LIN {X 0,Y 233.314,Z 747.017,A -85,B 0,C 180,E1 -22157.757,E2 -22157.757} C_VEL
LIN {X 0,Y 234.312,Z 748.351,A -85,B 0,C 180,E1 -22158.64,E2 -22158.64} C_VEL
LIN {X 0,Y 237.807,Z 753.166,A -85,B 0,C 180,E1 -22161.415,E2 -22161.415} C_VEL
LIN {X 0,Y 240.661,Z 757.385,A -85,B 0,C 180,E1 -22163.417,E2 -22163.417} C_VEL
LIN {X 0,Y 245.508,Z 764.562,A -85,B 0,C 180,E1 -22166.397,E2 -22166.397} C_VEL
LIN {X 0,Y 250.605,Z 772.878,A -85,B 0,C 180,E1 -22169.16,E2 -22169.16} C_VEL
LIN {X 0,Y 260.08,Z 786.969,A -85,B 0,C 180,E1 -22173.436,E2 -22173.436} C_VEL
LIN {X 0,Y 267.5,Z 795.645,A -85,B 0,C 180,E1 -22176.179,E2 -22176.179} C_VEL
LIN {X 0,Y 274.994,Z 803.198,A -85,B 0,C 180,E1 -22178.59,E2 -22178.59} C_VEL
LIN {X 0,Y 289.384,Z 815.503,A -85,B 0,C 180,E1 -22182.579,E2 -22182.579} C_VEL
LIN {X 0,Y 297.408,Z 822.094,A -85,B 0,C 180,E1 -22184.884,E2 -22184.884} C_VEL
LIN {X 0,Y 304.266,Z 827.849,A -85,B 0,C 180,E1 -22187.056,E2 -22187.056} C_VEL
LIN {X 0,Y 310.212,Z 832.821,A -85,B 0,C 180,E1 -22189.111,E2 -22189.111} C_VEL
LIN {X 0,Y 316.754,Z 838.584,A -85,B 0,C 180,E1 -22191.56,E2 -22191.56} C_VEL
LIN {X 0,Y 321.993,Z 842.915,A -85,B 0,C 180,E1 -22193.61,E2 -22193.61} C_VEL
LIN {X 0,Y 327.654,Z 847.59,A -85,B 0,C 180,E1 -22195.919,E2 -22195.919} C_VEL
LIN {X 0,Y 333.978,Z 853.067,A -85,B 0,C 180,E1 -22198.672,E2 -22198.672} C_VEL
LIN {X 0,Y 338.981,Z 856.943,A -85,B 0,C 180,E1 -22200.959,E2 -22200.959} C_VEL
LIN {X 0,Y 343.44,Z 860.757,A -85,B 0,C 180,E1 -22203.147,E2 -22203.147} C_VEL
LIN {X 0,Y 347.97,Z 863.872,A -85,B 0,C 180,E1 -22205.496,E2 -22205.496} C_VEL
LIN {X 0,Y 352.286,Z 867.651,A -85,B 0,C 180,E1 -22208.002,E2 -22208.002} C_VEL
LIN {X 0,Y 356.283,Z 870.579,A -85,B 0,C 180,E1 -22210.538,E2 -22210.538} C_VEL
LIN {X 0,Y 359.499,Z 872.581,A -85,B 0,C 180,E1 -22212.766,E2 -22212.766} C_VEL
LIN {X 0,Y 362.492,Z 875.444,A -85,B 0,C 180,E1 -22215.247,E2 -22215.247} C_VEL
LIN {X 0,Y 365.132,Z 877.452,A -85,B 0,C 180,E1 -22217.777,E2 -22217.777} C_VEL
LIN {X 0,Y 367.207,Z 878.655,A -85,B 0,C 180,E1 -22220.082,E2 -22220.082} C_VEL
LIN {X 0,Y 368.794,Z 879.391,A -85,B 0,C 180,E1 -22222.334,E2 -22222.334} C_VEL
LIN {X 0,Y 369.977,Z 879.911,A -85,B 0,C 180,E1 -22224.55,E2 -22224.55} C_VEL
LIN {X 0,Y 370.787,Z 880.342,A -85,B 0,C 180,E1 -22226.74,E2 -22226.74} C_VEL
LIN {X 0,Y 371.141,Z 880.49,A -85,B 0,C 180,E1 -22228.915,E2 -22228.915} C_VEL
LIN {X 0,Y 371.14,Z 880.491,A -85,B 0,C 180,E1 -22231.085,E2 -22231.085} C_VEL
LIN {X 0,Y 370.787,Z 880.343,A -85,B 0,C 180,E1 -22233.26,E2 -22233.26} C_VEL
LIN {X 0,Y 369.977,Z 879.915,A -85,B 0,C 180,E1 -22235.45,E2 -22235.45} C_VEL
LIN {X 0,Y 368.777,Z 879.363,A -85,B 0,C 180,E1 -22237.7,E2 -22237.7} C_VEL
LIN {X 0,Y 366.736,Z 878.408,A -85,B 0,C 180,E1 -22240.449,E2 -22240.449} C_VEL
LIN {X 0,Y 364.408,Z 876.944,A -85,B 0,C 180,E1 -22242.986,E2 -22242.986} C_VEL
LIN {X 0,Y 361.479,Z 874.571,A -85,B 0,C 180,E1 -22245.627,E2 -22245.627} C_VEL
LIN {X 0,Y 358.848,Z 871.974,A -85,B 0,C 180,E1 -22247.72,E2 -22247.72} C_VEL
LIN {X 0,Y 355.4,Z 869.953,A -85,B 0,C 180,E1 -22250.056,E2 -22250.056} C_VEL
LIN {X 0,Y 351.316,Z 866.844,A -85,B 0,C 180,E1 -22252.572,E2 -22252.572} C_VEL
LIN {X 0,Y 347.804,Z 863.747,A -85,B 0,C 180,E1 -22254.592,E2 -22254.592} C_VEL
LIN {X 0,Y 342.734,Z 860.245,A -85,B 0,C 180,E1 -22257.204,E2 -22257.204} C_VEL
LIN {X 0,Y 337.022,Z 855.328,A -85,B 0,C 180,E1 -22259.96,E2 -22259.96} C_VEL
LIN {X 0,Y 331.892,Z 851.318,A -85,B 0,C 180,E1 -22262.255,E2 -22262.255} C_VEL
LIN {X 0,Y 326.884,Z 847.01,A -85,B 0,C 180,E1 -22264.4,E2 -22264.4} C_VEL
LIN {X 0,Y 321.053,Z 842.045,A -85,B 0,C 180,E1 -22266.767,E2 -22266.767} C_VEL
LIN {X 0,Y 313.987,Z 836.199,A -85,B 0,C 180,E1 -22269.498,E2 -22269.498} C_VEL
LIN {X 0,Y 307.168,Z 830.349,A -85,B 0,C 180,E1 -22271.968,E2 -22271.968} C_VEL
LIN {X 0,Y 300.834,Z 824.92,A -85,B 0,C 180,E1 -22274.041,E2 -22274.041} C_VEL
LIN {X 0,Y 294.494,Z 819.582,A -85,B 0,C 180,E1 -22275.97,E2 -22275.97} C_VEL
LIN {X 0,Y 286.718,Z 813.265,A -85,B 0,C 180,E1 -22278.147,E2 -22278.147} C_VEL
LIN {X 0,Y 276.516,Z 804.475,A -85,B 0,C 180,E1 -22280.962,E2 -22280.962} C_VEL
LIN {X 0,Y 269.019,Z 797.351,A -85,B 0,C 180,E1 -22283.303,E2 -22283.303} C_VEL
LIN {X 0,Y 259.248,Z 785.918,A -85,B 0,C 180,E1 -22286.898,E2 -22286.898} C_VEL
LIN {X 0,Y 247.028,Z 766.992,A -85,B 0,C 180,E1 -22292.742,E2 -22292.742} C_VEL
LIN {X 0,Y 241.698,Z 758.869,A -85,B 0,C 180,E1 -22295.909,E2 -22295.909} C_VEL
LIN {X 0,Y 238.957,Z 754.892,A -85,B 0,C 180,E1 -22297.749,E2 -22297.749} C_VEL
LIN {X 0,Y 236.64,Z 751.543,A -85,B 0,C 180,E1 -22299.463,E2 -22299.463} C_VEL
LIN {X 0,Y 233.435,Z 747.121,A -85,B 0,C 180,E1 -22302.139,E2 -22302.139} C_VEL
LIN {X 0,Y 230.685,Z 743.267,A -85,B 0,C 180,E1 -22304.879,E2 -22304.879} C_VEL
LIN {X 0,Y 230.017,Z 742.388,A -85,B 0,C 180,E1 -22305.626,E2 -22305.626} C_VEL
LIN {X 0,Y 227.655,Z 739.605,A -85,B 0,C 180,E1 -22308.65,E2 -22308.65} C_VEL
LIN {X 0,Y 226.765,Z 737.637,A -85,B 0,C 180,E1 -22310.215,E2 -22310.215} C_VEL
LIN {X 0,Y 224.026,Z 734.193,A -85,B 0,C 180,E1 -22320,E2 -22320} C_VEL
LIN {X 0,Y 226.883,Z 737.813,A -85,B 0,C 180,E1 -22329.585,E2 -22329.585} C_VEL
LIN {X 0,Y 228.698,Z 741.176,A -85,B 0,C 180,E1 -22332.423,E2 -22332.423} C_VEL
LIN {X 0,Y 230.599,Z 743.15,A -85,B 0,C 180,E1 -22334.619,E2 -22334.619} C_VEL
LIN {X 0,Y 233.265,Z 746.992,A -85,B 0,C 180,E1 -22337.309,E2 -22337.309} C_VEL
LIN {X 0,Y 234.487,Z 748.68,A -85,B 0,C 180,E1 -22338.391,E2 -22338.391} C_VEL
LIN {X 0,Y 237.725,Z 753.072,A -85,B 0,C 180,E1 -22340.949,E2 -22340.949} C_VEL
LIN {X 0,Y 240.892,Z 757.691,A -85,B 0,C 180,E1 -22343.16,E2 -22343.16} C_VEL
LIN {X 0,Y 245.663,Z 764.824,A -85,B 0,C 180,E1 -22346.08,E2 -22346.08} C_VEL
LIN {X 0,Y 250.2,Z 773.785,A -85,B 0,C 180,E1 -22348.638,E2 -22348.638} C_VEL
LIN {X 0,Y 254.973,Z 784.136,A -85,B 0,C 180,E1 -22351.084,E2 -22351.084} C_VEL
LIN {X 0,Y 259.68,Z 795.604,A -85,B 0,C 180,E1 -22353.32,E2 -22353.32} C_VEL
LIN {X 0,Y 252.558,Z 888.891,A -85,B 0,C 180,E1 -22355.604,E2 -22355.604} C_VEL
LIN {X 0,Y 250.81,Z 902.408,A -85,B 0,C 180,E1 -22356.075,E2 -22356.075} C_VEL
LIN {X 0,Y 248.59,Z 914.617,A -85,B 0,C 180,E1 -22356.608,E2 -22356.608} C_VEL
LIN {X 0,Y 245.71,Z 927.15,A -85,B 0,C 180,E1 -22357.298,E2 -22357.298} C_VEL
LIN {X 0,Y 243.03,Z 937.334,A -85,B 0,C 180,E1 -22358.001,E2 -22358.001} C_VEL
LIN {X 0,Y 238.986,Z 950.564,A -85,B 0,C 180,E1 -22359.14,E2 -22359.14} C_VEL
LIN {X 0,Y 235.019,Z 961.857,A -85,B 0,C 180,E1 -22360.312,E2 -22360.312} C_VEL
LIN {X 0,Y 230.1,Z 974.284,A -85,B 0,C 180,E1 -22361.886,E2 -22361.886} C_VEL
LIN {X 0,Y 226.127,Z 983.479,A -85,B 0,C 180,E1 -22363.256,E2 -22363.256} C_VEL
LIN {X 0,Y 220.297,Z 995.568,A -85,B 0,C 180,E1 -22365.426,E2 -22365.426} C_VEL
LIN {X 0,Y 215.559,Z 1004.833,A -85,B 0,C 180,E1 -22367.429,E2 -22367.429} C_VEL
LIN {X 0,Y 213.299,Z 1009.008,A -85,B 0,C 180,E1 -22368.464,E2 -22368.464} C_VEL
LIN {X 0,Y 210.589,Z 1013.057,A -85,B 0,C 180,E1 -22369.393,E2 -22369.393} C_VEL
LIN {X 0,Y 199.902,Z 1024.022,A -85,B 0,C 180,E1 -22371.945,E2 -22371.945} C_VEL
LIN {X 0,Y 196.93,Z 1027.478,A -85,B 0,C 180,E1 -22373.029,E2 -22373.029} C_VEL
LIN {X 0,Y 196.166,Z 1028.612,A -85,B 0,C 180,E1 -22373.441,E2 -22373.441} C_VEL
LIN {X 0,Y 190.245,Z 1037.906,A -85,B 0,C 180,E1 -22377.613,E2 -22377.613} C_VEL
LIN {X 0,Y 185.606,Z 1045.172,A -85,B 0,C 180,E1 -22381.751,E2 -22381.751} C_VEL
LIN {X 0,Y 182.728,Z 1049.828,A -85,B 0,C 180,E1 -22384.972,E2 -22384.972} C_VEL
LIN {X 0,Y 179.742,Z 1054.936,A -85,B 0,C 180,E1 -22389.397,E2 -22389.397} C_VEL
LIN {X 0,Y 177.665,Z 1058.948,A -85,B 0,C 180,E1 -22393.925,E2 -22393.925} C_VEL
LIN {X 0,Y 176.412,Z 1061.919,A -85,B 0,C 180,E1 -22398.511,E2 -22398.511} C_VEL
LIN {X 0,Y 176.09,Z 1063.115,A -85,B 0,C 180,E1 -22400.814,E2 -22400.814} C_VEL
LIN {X 0,Y 175.876,Z 1064.6,A -85,B 0,C 180,E1 -22405.416,E2 -22405.416} C_VEL
LIN {X 0,Y 176.077,Z 1065.1,A -85,B 0,C 180,E1 -22410,E2 -22410} C_VEL
LIN {X 0,Y 175.876,Z 1064.6,A -85,B 0,C 180,E1 -22414.584,E2 -22414.584} C_VEL
LIN {X 0,Y 176.09,Z 1063.115,A -85,B 0,C 180,E1 -22419.186,E2 -22419.186} C_VEL
LIN {X 0,Y 176.885,Z 1060.628,A -85,B 0,C 180,E1 -22423.791,E2 -22423.791} C_VEL
LIN {X 0,Y 178.603,Z 1057.119,A -85,B 0,C 180,E1 -22428.348,E2 -22428.348} C_VEL
LIN {X 0,Y 181.11,Z 1052.53,A -85,B 0,C 180,E1 -22432.833,E2 -22432.833} C_VEL
LIN {X 0,Y 184.609,Z 1046.796,A -85,B 0,C 180,E1 -22437.182,E2 -22437.182} C_VEL
LIN {X 0,Y 188.445,Z 1040.648,A -85,B 0,C 180,E1 -22440.931,E2 -22440.931} C_VEL
LIN {X 0,Y 192.903,Z 1033.696,A -85,B 0,C 180,E1 -22444.381,E2 -22444.381} C_VEL
LIN {X 0,Y 197.376,Z 1026.716,A -85,B 0,C 180,E1 -22447.251,E2 -22447.251} C_VEL
LIN {X 0,Y 202.161,Z 1018.842,A -85,B 0,C 180,E1 -22449.984,E2 -22449.984} C_VEL
LIN {X 0,Y 207.527,Z 1009.64,A -85,B 0,C 180,E1 -22452.632,E2 -22452.632} C_VEL
LIN {X 0,Y 212.222,Z 1001.074,A -85,B 0,C 180,E1 -22454.725,E2 -22454.725} C_VEL
LIN {X 0,Y 218.392,Z 989.22,A -85,B 0,C 180,E1 -22457.062,E2 -22457.062} C_VEL
LIN {X 0,Y 223.032,Z 979.459,A -85,B 0,C 180,E1 -22458.682,E2 -22458.682} C_VEL
LIN {X 0,Y 228.172,Z 967.399,A -85,B 0,C 180,E1 -22460.355,E2 -22460.355} C_VEL
LIN {X 0,Y 232.807,Z 955.383,A -85,B 0,C 180,E1 -22461.709,E2 -22461.709} C_VEL
LIN {X 0,Y 236.912,Z 943.069,A -85,B 0,C 180,E1 -22462.866,E2 -22462.866} C_VEL
LIN {X 0,Y 240.525,Z 930.531,A -85,B 0,C 180,E1 -22463.82,E2 -22463.82} C_VEL
LIN {X 0,Y 243.814,Z 917.215,A -85,B 0,C 180,E1 -22464.594,E2 -22464.594} C_VEL
LIN {X 0,Y 246.415,Z 903.799,A -85,B 0,C 180,E1 -22465.206,E2 -22465.206} C_VEL
LIN {X 0,Y 248.222,Z 891.368,A -85,B 0,C 180,E1 -22465.638,E2 -22465.638} C_VEL
LIN {X 0,Y 250.423,Z 865.327,A -85,B 0,C 180,E1 -22466.332,E2 -22466.332} C_VEL
LIN {X 0,Y 255.581,Z 798.34,A -85,B 0,C 180,E1 -22467.952,E2 -22467.952} C_VEL
LIN {X 0,Y 250.489,Z 785.853,A -85,B 0,C 180,E1 -22470.549,E2 -22470.549} C_VEL
LIN {X 0,Y 245.29,Z 774.673,A -85,B 0,C 180,E1 -22473.462,E2 -22473.462} C_VEL
LIN {X 0,Y 242.766,Z 769.848,A -85,B 0,C 180,E1 -22474.996,E2 -22474.996} C_VEL
LIN {X 0,Y 237.598,Z 761.907,A -85,B 0,C 180,E1 -22478.414,E2 -22478.414} C_VEL
LIN {X 0,Y 234.666,Z 757.732,A -85,B 0,C 180,E1 -22480.651,E2 -22480.651} C_VEL
LIN {X 0,Y 231.946,Z 753.775,A -85,B 0,C 180,E1 -22483.044,E2 -22483.044} C_VEL
LIN {X 0,Y 229.379,Z 750.136,A -85,B 0,C 180,E1 -22485.698,E2 -22485.698} C_VEL
LIN {X 0,Y 228.452,Z 749.019,A -85,B 0,C 180,E1 -22486.773,E2 -22486.773} C_VEL
LIN {X 0,Y 226.154,Z 745.723,A -85,B 0,C 180,E1 -22490.045,E2 -22490.045} C_VEL
LIN {X 0,Y 225.635,Z 744.532,A -85,B 0,C 180,E1 -22491.04,E2 -22491.04} C_VEL
LIN {X 0,Y 223.158,Z 741.269,A -85,B 0,C 180,E1 -22500,E2 -22500} C_VEL
LIN {X 0,Y 225.774,Z 744.727,A -85,B 0,C 180,E1 -22509.62,E2 -22509.62} C_VEL
LIN {X 0,Y 227.537,Z 748.005,A -85,B 0,C 180,E1 -22512.486,E2 -22512.486} C_VEL
LIN {X 0,Y 229.424,Z 750.128,A -85,B 0,C 180,E1 -22514.752,E2 -22514.752} C_VEL
LIN {X 0,Y 231.992,Z 753.846,A -85,B 0,C 180,E1 -22517.408,E2 -22517.408} C_VEL
LIN {X 0,Y 236.02,Z 759.62,A -85,B 0,C 180,E1 -22520.821,E2 -22520.821} C_VEL
LIN {X 0,Y 238.713,Z 763.657,A -85,B 0,C 180,E1 -22522.788,E2 -22522.788} C_VEL
LIN {X 0,Y 243.216,Z 770.59,A -85,B 0,C 180,E1 -22525.686,E2 -22525.686} C_VEL
LIN {X 0,Y 247.32,Z 777.402,A -85,B 0,C 180,E1 -22528.031,E2 -22528.031} C_VEL
LIN {X 0,Y 257.171,Z 792.629,A -85,B 0,C 180,E1 -22532.723,E2 -22532.723} C_VEL
LIN {X 0,Y 264.837,Z 801.783,A -85,B 0,C 180,E1 -22535.659,E2 -22535.659} C_VEL
LIN {X 0,Y 272.121,Z 809.233,A -85,B 0,C 180,E1 -22538.075,E2 -22538.075} C_VEL
LIN {X 0,Y 288.085,Z 822.884,A -85,B 0,C 180,E1 -22542.552,E2 -22542.552} C_VEL
LIN {X 0,Y 294.539,Z 828.106,A -85,B 0,C 180,E1 -22544.385,E2 -22544.385} C_VEL
LIN {X 0,Y 302.586,Z 834.742,A -85,B 0,C 180,E1 -22546.864,E2 -22546.864} C_VEL
LIN {X 0,Y 308.947,Z 839.935,A -85,B 0,C 180,E1 -22549.028,E2 -22549.028} C_VEL
LIN {X 0,Y 315.11,Z 845.372,A -85,B 0,C 180,E1 -22551.316,E2 -22551.316} C_VEL
LIN {X 0,Y 320.226,Z 849.618,A -85,B 0,C 180,E1 -22553.309,E2 -22553.309} C_VEL
LIN {X 0,Y 326.087,Z 854.351,A -85,B 0,C 180,E1 -22555.675,E2 -22555.675} C_VEL
LIN {X 0,Y 332.373,Z 859.782,A -85,B 0,C 180,E1 -22558.384,E2 -22558.384} C_VEL
LIN {X 0,Y 337.741,Z 863.932,A -85,B 0,C 180,E1 -22560.821,E2 -22560.821} C_VEL
LIN {X 0,Y 342.17,Z 867.657,A -85,B 0,C 180,E1 -22562.977,E2 -22562.977} C_VEL
LIN {X 0,Y 346.893,Z 870.883,A -85,B 0,C 180,E1 -22565.415,E2 -22565.415} C_VEL
LIN {X 0,Y 350.998,Z 874.506,A -85,B 0,C 180,E1 -22567.787,E2 -22567.787} C_VEL
LIN {X 0,Y 355.296,Z 877.615,A -85,B 0,C 180,E1 -22570.482,E2 -22570.482} C_VEL
LIN {X 0,Y 358.403,Z 879.535,A -85,B 0,C 180,E1 -22572.609,E2 -22572.609} C_VEL
LIN {X 0,Y 361.553,Z 882.503,A -85,B 0,C 180,E1 -22575.208,E2 -22575.208} C_VEL
LIN {X 0,Y 364.226,Z 884.477,A -85,B 0,C 180,E1 -22577.746,E2 -22577.746} C_VEL
LIN {X 0,Y 366.31,Z 885.676,A -85,B 0,C 180,E1 -22580.057,E2 -22580.057} C_VEL
LIN {X 0,Y 368.088,Z 886.536,A -85,B 0,C 180,E1 -22582.622,E2 -22582.622} C_VEL
LIN {X 0,Y 369.185,Z 887.01,A -85,B 0,C 180,E1 -22584.705,E2 -22584.705} C_VEL
LIN {X 0,Y 369.923,Z 887.364,A -85,B 0,C 180,E1 -22586.733,E2 -22586.733} C_VEL
LIN {X 0,Y 370.274,Z 887.537,A -85,B 0,C 180,E1 -22588.912,E2 -22588.912} C_VEL
LIN {X 0,Y 370.274,Z 887.537,A -85,B 0,C 180,E1 -22591.088,E2 -22591.088} C_VEL
LIN {X 0,Y 369.923,Z 887.366,A -85,B 0,C 180,E1 -22593.267,E2 -22593.267} C_VEL
LIN {X 0,Y 369.102,Z 886.957,A -85,B 0,C 180,E1 -22595.463,E2 -22595.463} C_VEL
LIN {X 0,Y 367.916,Z 886.416,A -85,B 0,C 180,E1 -22597.684,E2 -22597.684} C_VEL
LIN {X 0,Y 366.033,Z 885.567,A -85,B 0,C 180,E1 -22600.248,E2 -22600.248} C_VEL
LIN {X 0,Y 363.695,Z 884.127,A -85,B 0,C 180,E1 -22602.829,E2 -22602.829} C_VEL
LIN {X 0,Y 360.935,Z 881.961,A -85,B 0,C 180,E1 -22605.32,E2 -22605.32} C_VEL
LIN {X 0,Y 357.428,Z 878.795,A -85,B 0,C 180,E1 -22608.078,E2 -22608.078} C_VEL
LIN {X 0,Y 353.746,Z 876.555,A -85,B 0,C 180,E1 -22610.533,E2 -22610.533} C_VEL
LIN {X 0,Y 349.616,Z 873.308,A -85,B 0,C 180,E1 -22613.048,E2 -22613.048} C_VEL
LIN {X 0,Y 346.144,Z 870.378,A -85,B 0,C 180,E1 -22614.975,E2 -22614.975} C_VEL
LIN {X 0,Y 341.142,Z 866.913,A -85,B 0,C 180,E1 -22617.52,E2 -22617.52} C_VEL
LIN {X 0,Y 335.607,Z 862.146,A -85,B 0,C 180,E1 -22620.17,E2 -22620.17} C_VEL
LIN {X 0,Y 330.383,Z 858.142,A -85,B 0,C 180,E1 -22622.485,E2 -22622.485} C_VEL
LIN {X 0,Y 325.298,Z 853.789,A -85,B 0,C 180,E1 -22624.644,E2 -22624.644} C_VEL
LIN {X 0,Y 319.257,Z 848.709,A -85,B 0,C 180,E1 -22627.084,E2 -22627.084} C_VEL
LIN {X 0,Y 312.11,Z 842.822,A -85,B 0,C 180,E1 -22629.816,E2 -22629.816} C_VEL
LIN {X 0,Y 306.006,Z 837.612,A -85,B 0,C 180,E1 -22631.993,E2 -22631.993} C_VEL
LIN {X 0,Y 299.443,Z 832.053,A -85,B 0,C 180,E1 -22634.122,E2 -22634.122} C_VEL
LIN {X 0,Y 293.478,Z 827.213,A -85,B 0,C 180,E1 -22635.922,E2 -22635.922} C_VEL
LIN {X 0,Y 285.835,Z 821.012,A -85,B 0,C 180,E1 -22638.058,E2 -22638.058} C_VEL
LIN {X 0,Y 273.861,Z 810.739,A -85,B 0,C 180,E1 -22641.398,E2 -22641.398} C_VEL
LIN {X 0,Y 265.99,Z 803.077,A -85,B 0,C 180,E1 -22643.935,E2 -22643.935} C_VEL
LIN {X 0,Y 258.419,Z 794.171,A -85,B 0,C 180,E1 -22646.769,E2 -22646.769} C_VEL
LIN {X 0,Y 250.96,Z 783.524,A -85,B 0,C 180,E1 -22650.085,E2 -22650.085} C_VEL
LIN {X 0,Y 244.766,Z 773.082,A -85,B 0,C 180,E1 -22653.402,E2 -22653.402} C_VEL
LIN {X 0,Y 239.513,Z 764.889,A -85,B 0,C 180,E1 -22656.664,E2 -22656.664} C_VEL
LIN {X 0,Y 236.595,Z 760.528,A -85,B 0,C 180,E1 -22658.736,E2 -22658.736} C_VEL
LIN {X 0,Y 234.721,Z 757.783,A -85,B 0,C 180,E1 -22660.202,E2 -22660.202} C_VEL
LIN {X 0,Y 231.992,Z 753.847,A -85,B 0,C 180,E1 -22662.592,E2 -22662.592} C_VEL
LIN {X 0,Y 229.243,Z 749.811,A -85,B 0,C 180,E1 -22665.463,E2 -22665.463} C_VEL
LIN {X 0,Y 226.367,Z 746.177,A -85,B 0,C 180,E1 -22669.265,E2 -22669.265} C_VEL
LIN {X 0,Y 225.733,Z 744.626,A -85,B 0,C 180,E1 -22670.462,E2 -22670.462} C_VEL
LIN {X 0,Y 223.159,Z 741.256,A -85,B 0,C 180,E1 -22680,E2 -22680} C_VEL
LIN {X 0,Y 225.813,Z 744.825,A -85,B 0,C 180,E1 -22689.292,E2 -22689.292} C_VEL
LIN {X 0,Y 227.667,Z 748.185,A -85,B 0,C 180,E1 -22692.253,E2 -22692.253} C_VEL
LIN {X 0,Y 229.292,Z 749.948,A -85,B 0,C 180,E1 -22694.194,E2 -22694.194} C_VEL
LIN {X 0,Y 231.941,Z 753.818,A -85,B 0,C 180,E1 -22696.957,E2 -22696.957} C_VEL
LIN {X 0,Y 236.031,Z 759.636,A -85,B 0,C 180,E1 -22700.423,E2 -22700.423} C_VEL
LIN {X 0,Y 239.216,Z 764.433,A -85,B 0,C 180,E1 -22702.728,E2 -22702.728} C_VEL
LIN {X 0,Y 243.707,Z 771.408,A -85,B 0,C 180,E1 -22705.574,E2 -22705.574} C_VEL
LIN {X 0,Y 248.263,Z 781.006,A -85,B 0,C 180,E1 -22708.248,E2 -22708.248} C_VEL
LIN {X 0,Y 252.005,Z 789.421,A -85,B 0,C 180,E1 -22710.248,E2 -22710.248} C_VEL
LIN {X 0,Y 255.584,Z 798.31,A -85,B 0,C 180,E1 -22712.047,E2 -22712.047} C_VEL
LIN {X 0,Y 248.488,Z 888.695,A -85,B 0,C 180,E1 -22714.272,E2 -22714.272} C_VEL
LIN {X 0,Y 246.671,Z 902.327,A -85,B 0,C 180,E1 -22714.745,E2 -22714.745} C_VEL
LIN {X 0,Y 244.361,Z 914.712,A -85,B 0,C 180,E1 -22715.288,E2 -22715.288} C_VEL
LIN {X 0,Y 241.462,Z 926.944,A -85,B 0,C 180,E1 -22715.954,E2 -22715.954} C_VEL
LIN {X 0,Y 238.714,Z 937.128,A -85,B 0,C 180,E1 -22716.655,E2 -22716.655} C_VEL
LIN {X 0,Y 234.552,Z 950.358,A -85,B 0,C 180,E1 -22717.79,E2 -22717.79} C_VEL
LIN {X 0,Y 230.474,Z 961.651,A -85,B 0,C 180,E1 -22718.962,E2 -22718.962} C_VEL
LIN {X 0,Y 225.375,Z 974.077,A -85,B 0,C 180,E1 -22720.529,E2 -22720.529} C_VEL
LIN {X 0,Y 220.919,Z 984.023,A -85,B 0,C 180,E1 -22722.036,E2 -22722.036} C_VEL
LIN {X 0,Y 215.272,Z 995.361,A -85,B 0,C 180,E1 -22724.093,E2 -22724.093} C_VEL
LIN {X 0,Y 210.328,Z 1004.625,A -85,B 0,C 180,E1 -22726.105,E2 -22726.105} C_VEL
LIN {X 0,Y 204.802,Z 1014.354,A -85,B 0,C 180,E1 -22728.657,E2 -22728.657} C_VEL
LIN {X 0,Y 199.738,Z 1022.876,A -85,B 0,C 180,E1 -22731.352,E2 -22731.352} C_VEL
LIN {X 0,Y 196.166,Z 1028.612,A -85,B 0,C 180,E1 -22733.441,E2 -22733.441} C_VEL
LIN {X 0,Y 193.542,Z 1031.931,A -85,B 0,C 180,E1 -22734.657,E2 -22734.657} C_VEL
LIN {X 0,Y 187.783,Z 1037.033,A -85,B 0,C 180,E1 -22736.543,E2 -22736.543} C_VEL
LIN {X 0,Y 182.161,Z 1041.648,A -85,B 0,C 180,E1 -22738.631,E2 -22738.631} C_VEL
LIN {X 0,Y 179.814,Z 1044.194,A -85,B 0,C 180,E1 -22740.145,E2 -22740.145} C_VEL
LIN {X 0,Y 176.205,Z 1049.619,A -85,B 0,C 180,E1 -22743.977,E2 -22743.977} C_VEL
LIN {X 0,Y 173.004,Z 1054.727,A -85,B 0,C 180,E1 -22748.555,E2 -22748.555} C_VEL
LIN {X 0,Y 170.757,Z 1058.74,A -85,B 0,C 180,E1 -22753.256,E2 -22753.256} C_VEL
LIN {X 0,Y 169.389,Z 1061.712,A -85,B 0,C 180,E1 -22758.027,E2 -22758.027} C_VEL
LIN {X 0,Y 169.037,Z 1062.908,A -85,B 0,C 180,E1 -22760.427,E2 -22760.427} C_VEL
LIN {X 0,Y 168.771,Z 1064.393,A -85,B 0,C 180,E1 -22765.223,E2 -22765.223} C_VEL
LIN {X 0,Y 168.985,Z 1064.894,A -85,B 0,C 180,E1 -22770,E2 -22770} C_VEL
LIN {X 0,Y 168.771,Z 1064.393,A -85,B 0,C 180,E1 -22774.777,E2 -22774.777} C_VEL
LIN {X 0,Y 169.037,Z 1062.908,A -85,B 0,C 180,E1 -22779.573,E2 -22779.573} C_VEL
LIN {X 0,Y 169.932,Z 1060.421,A -85,B 0,C 180,E1 -22784.367,E2 -22784.367} C_VEL
LIN {X 0,Y 172.371,Z 1055.781,A -85,B 0,C 180,E1 -22790.32,E2 -22790.32} C_VEL
LIN {X 0,Y 174.477,Z 1052.321,A -85,B 0,C 180,E1 -22793.753,E2 -22793.753} C_VEL
LIN {X 0,Y 178.209,Z 1046.586,A -85,B 0,C 180,E1 -22798.244,E2 -22798.244} C_VEL
LIN {X 0,Y 181.943,Z 1040.963,A -85,B 0,C 180,E1 -22801.809,E2 -22801.809} C_VEL
LIN {X 0,Y 186.999,Z 1033.488,A -85,B 0,C 180,E1 -22805.628,E2 -22805.628} C_VEL
LIN {X 0,Y 191.712,Z 1026.508,A -85,B 0,C 180,E1 -22808.549,E2 -22808.549} C_VEL
LIN {X 0,Y 197.039,Z 1018.099,A -85,B 0,C 180,E1 -22811.493,E2 -22811.493} C_VEL
LIN {X 0,Y 202.306,Z 1009.432,A -85,B 0,C 180,E1 -22814.009,E2 -22814.009} C_VEL
LIN {X 0,Y 207.177,Z 1000.866,A -85,B 0,C 180,E1 -22816.124,E2 -22816.124} C_VEL
LIN {X 0,Y 213.579,Z 989.013,A -85,B 0,C 180,E1 -22818.468,E2 -22818.468} C_VEL
LIN {X 0,Y 219.103,Z 977.608,A -85,B 0,C 180,E1 -22820.337,E2 -22820.337} C_VEL
LIN {X 0,Y 223.691,Z 967.193,A -85,B 0,C 180,E1 -22821.761,E2 -22821.761} C_VEL
LIN {X 0,Y 228.45,Z 955.176,A -85,B 0,C 180,E1 -22823.115,E2 -22823.115} C_VEL
LIN {X 0,Y 232.675,Z 942.862,A -85,B 0,C 180,E1 -22824.267,E2 -22824.267} C_VEL
LIN {X 0,Y 236.395,Z 930.325,A -85,B 0,C 180,E1 -22825.212,E2 -22825.212} C_VEL
LIN {X 0,Y 239.715,Z 917.23,A -85,B 0,C 180,E1 -22825.969,E2 -22825.969} C_VEL
LIN {X 0,Y 242.343,Z 904.144,A -85,B 0,C 180,E1 -22826.564,E2 -22826.564} C_VEL
LIN {X 0,Y 244.279,Z 891.236,A -85,B 0,C 180,E1 -22827.01,E2 -22827.01} C_VEL
LIN {X 0,Y 246.527,Z 865.511,A -85,B 0,C 180,E1 -22827.696,E2 -22827.696} C_VEL
LIN {X 0,Y 251.613,Z 801.254,A -85,B 0,C 180,E1 -22829.255,E2 -22829.255} C_VEL
LIN {X 0,Y 247.239,Z 790.194,A -85,B 0,C 180,E1 -22831.641,E2 -22831.641} C_VEL
LIN {X 0,Y 242.734,Z 780.198,A -85,B 0,C 180,E1 -22834.316,E2 -22834.316} C_VEL
LIN {X 0,Y 240.666,Z 776.063,A -85,B 0,C 180,E1 -22835.639,E2 -22835.639} C_VEL
LIN {X 0,Y 235.745,Z 768.262,A -85,B 0,C 180,E1 -22839.038,E2 -22839.038} C_VEL
LIN {X 0,Y 232.933,Z 764.121,A -85,B 0,C 180,E1 -22841.285,E2 -22841.285} C_VEL
LIN {X 0,Y 230.293,Z 760.257,A -85,B 0,C 180,E1 -22843.717,E2 -22843.717} C_VEL
LIN {X 0,Y 227.459,Z 756.051,A -85,B 0,C 180,E1 -22846.885,E2 -22846.885} C_VEL
LIN {X 0,Y 225.096,Z 752.736,A -85,B 0,C 180,E1 -22850.31,E2 -22850.31} C_VEL
LIN {X 0,Y 224.523,Z 751.444,A -85,B 0,C 180,E1 -22851.449,E2 -22851.449} C_VEL
LIN {X 0,Y 222.291,Z 748.326,A -85,B 0,C 180,E1 -22860,E2 -22860} C_VEL
LIN {X 0,Y 224.686,Z 751.646,A -85,B 0,C 180,E1 -22869.265,E2 -22869.265} C_VEL
LIN {X 0,Y 226.509,Z 755.031,A -85,B 0,C 180,E1 -22872.316,E2 -22872.316} C_VEL
LIN {X 0,Y 228.081,Z 756.866,A -85,B 0,C 180,E1 -22874.27,E2 -22874.27} C_VEL
LIN {X 0,Y 230.594,Z 760.591,A -85,B 0,C 180,E1 -22876.976,E2 -22876.976} C_VEL
LIN {X 0,Y 234.444,Z 766.337,A -85,B 0,C 180,E1 -22880.365,E2 -22880.365} C_VEL
LIN {X 0,Y 237.105,Z 770.479,A -85,B 0,C 180,E1 -22882.377,E2 -22882.377} C_VEL
LIN {X 0,Y 241.206,Z 777.012,A -85,B 0,C 180,E1 -22885.113,E2 -22885.113} C_VEL
LIN {X 0,Y 245.056,Z 783.616,A -85,B 0,C 180,E1 -22887.404,E2 -22887.404} C_VEL
LIN {X 0,Y 254.56,Z 798.622,A -85,B 0,C 180,E1 -22892.104,E2 -22892.104} C_VEL
LIN {X 0,Y 262.295,Z 808.008,A -85,B 0,C 180,E1 -22895.164,E2 -22895.164} C_VEL
LIN {X 0,Y 269.776,Z 815.705,A -85,B 0,C 180,E1 -22897.707,E2 -22897.707} C_VEL
LIN {X 0,Y 279.565,Z 824.256,A -85,B 0,C 180,E1 -22900.582,E2 -22900.582} C_VEL
LIN {X 0,Y 287.772,Z 830.912,A -85,B 0,C 180,E1 -22902.786,E2 -22902.786} C_VEL
LIN {X 0,Y 296.284,Z 837.838,A -85,B 0,C 180,E1 -22905.239,E2 -22905.239} C_VEL
LIN {X 0,Y 303.242,Z 843.656,A -85,B 0,C 180,E1 -22907.452,E2 -22907.452} C_VEL
LIN {X 0,Y 308.441,Z 847.879,A -85,B 0,C 180,E1 -22909.234,E2 -22909.234} C_VEL
LIN {X 0,Y 314.476,Z 852.966,A -85,B 0,C 180,E1 -22911.46,E2 -22911.46} C_VEL
LIN {X 0,Y 320.775,Z 858.24,A -85,B 0,C 180,E1 -22913.922,E2 -22913.922} C_VEL
LIN {X 0,Y 326.804,Z 863.111,A -85,B 0,C 180,E1 -22916.395,E2 -22916.395} C_VEL
LIN {X 0,Y 332.448,Z 867.833,A -85,B 0,C 180,E1 -22918.849,E2 -22918.849} C_VEL
LIN {X 0,Y 336.326,Z 870.763,A -85,B 0,C 180,E1 -22920.595,E2 -22920.595} C_VEL
LIN {X 0,Y 340.731,Z 874.471,A -85,B 0,C 180,E1 -22922.737,E2 -22922.737} C_VEL
LIN {X 0,Y 345.594,Z 877.77,A -85,B 0,C 180,E1 -22925.222,E2 -22925.222} C_VEL
LIN {X 0,Y 349.841,Z 881.444,A -85,B 0,C 180,E1 -22927.644,E2 -22927.644} C_VEL
LIN {X 0,Y 353.862,Z 884.354,A -85,B 0,C 180,E1 -22930.125,E2 -22930.125} C_VEL
LIN {X 0,Y 357.436,Z 886.623,A -85,B 0,C 180,E1 -22932.561,E2 -22932.561} C_VEL
LIN {X 0,Y 360.614,Z 889.558,A -85,B 0,C 180,E1 -22935.168,E2 -22935.168} C_VEL
LIN {X 0,Y 363.318,Z 891.523,A -85,B 0,C 180,E1 -22937.715,E2 -22937.715} C_VEL
LIN {X 0,Y 365.413,Z 892.699,A -85,B 0,C 180,E1 -22940.032,E2 -22940.032} C_VEL
LIN {X 0,Y 367.034,Z 893.462,A -85,B 0,C 180,E1 -22942.297,E2 -22942.297} C_VEL
LIN {X 0,Y 368.228,Z 893.99,A -85,B 0,C 180,E1 -22944.524,E2 -22944.524} C_VEL
LIN {X 0,Y 369.057,Z 894.41,A -85,B 0,C 180,E1 -22946.725,E2 -22946.725} C_VEL
LIN {X 0,Y 369.408,Z 894.583,A -85,B 0,C 180,E1 -22948.91,E2 -22948.91} C_VEL
LIN {X 0,Y 369.408,Z 894.583,A -85,B 0,C 180,E1 -22951.09,E2 -22951.09} C_VEL
LIN {X 0,Y 369.057,Z 894.411,A -85,B 0,C 180,E1 -22953.275,E2 -22953.275} C_VEL
LIN {X 0,Y 368.227,Z 894,A -85,B 0,C 180,E1 -22955.476,E2 -22955.476} C_VEL
LIN {X 0,Y 367.035,Z 893.459,A -85,B 0,C 180,E1 -22957.703,E2 -22957.703} C_VEL
LIN {X 0,Y 365.135,Z 892.608,A -85,B 0,C 180,E1 -22960.273,E2 -22960.273} C_VEL
LIN {X 0,Y 362.778,Z 891.174,A -85,B 0,C 180,E1 -22962.862,E2 -22962.862} C_VEL
LIN {X 0,Y 359.999,Z 889.016,A -85,B 0,C 180,E1 -22965.361,E2 -22965.361} C_VEL
LIN {X 0,Y 356.461,Z 885.822,A -85,B 0,C 180,E1 -22968.129,E2 -22968.129} C_VEL
LIN {X 0,Y 352.7,Z 883.574,A -85,B 0,C 180,E1 -22970.615,E2 -22970.615} C_VEL
LIN {X 0,Y 348.56,Z 880.353,A -85,B 0,C 180,E1 -22973.122,E2 -22973.122} C_VEL
LIN {X 0,Y 344.796,Z 877.211,A -85,B 0,C 180,E1 -22975.2,E2 -22975.2} C_VEL
LIN {X 0,Y 339.716,Z 873.723,A -85,B 0,C 180,E1 -22977.758,E2 -22977.758} C_VEL
LIN {X 0,Y 333.944,Z 868.824,A -85,B 0,C 180,E1 -22980.498,E2 -22980.498} C_VEL
LIN {X 0,Y 328.555,Z 864.671,A -85,B 0,C 180,E1 -22982.86,E2 -22982.86} C_VEL
LIN {X 0,Y 323.684,Z 860.542,A -85,B 0,C 180,E1 -22984.905,E2 -22984.905} C_VEL
LIN {X 0,Y 317.598,Z 855.486,A -85,B 0,C 180,E1 -22987.335,E2 -22987.335} C_VEL
LIN {X 0,Y 310.623,Z 849.835,A -85,B 0,C 180,E1 -22989.97,E2 -22989.97} C_VEL
LIN {X 0,Y 305.228,Z 845.182,A -85,B 0,C 180,E1 -22991.891,E2 -22991.891} C_VEL
LIN {X 0,Y 299.281,Z 840.31,A -85,B 0,C 180,E1 -22993.822,E2 -22993.822} C_VEL
LIN {X 0,Y 292.572,Z 834.895,A -85,B 0,C 180,E1 -22995.844,E2 -22995.844} C_VEL
LIN {X 0,Y 286.392,Z 829.888,A -85,B 0,C 180,E1 -22997.579,E2 -22997.579} C_VEL
LIN {X 0,Y 271.841,Z 817.603,A -85,B 0,C 180,E1 -23001.65,E2 -23001.65} C_VEL
LIN {X 0,Y 263.208,Z 809.067,A -85,B 0,C 180,E1 -23004.503,E2 -23004.503} C_VEL
LIN {X 0,Y 253.647,Z 797.42,A -85,B 0,C 180,E1 -23008.293,E2 -23008.293} C_VEL
LIN {X 0,Y 242.304,Z 778.835,A -85,B 0,C 180,E1 -23014.211,E2 -23014.211} C_VEL
LIN {X 0,Y 237.53,Z 771.135,A -85,B 0,C 180,E1 -23017.322,E2 -23017.322} C_VEL
LIN {X 0,Y 233.603,Z 764.922,A -85,B 0,C 180,E1 -23020.332,E2 -23020.332} C_VEL
LIN {X 0,Y 230.387,Z 760.362,A -85,B 0,C 180,E1 -23023.22,E2 -23023.22} C_VEL
LIN {X 0,Y 227.548,Z 756.086,A -85,B 0,C 180,E1 -23026.379,E2 -23026.379} C_VEL
LIN {X 0,Y 225.283,Z 753.124,A -85,B 0,C 180,E1 -23029.564,E2 -23029.564} C_VEL
LIN {X 0,Y 224.544,Z 751.49,A -85,B 0,C 180,E1 -23030.997,E2 -23030.997} C_VEL
LIN {X 0,Y 222.292,Z 748.319,A -85,B 0,C 180,E1 -23040,E2 -23040} C_VEL
LIN {X 0,Y 224.698,Z 751.68,A -85,B 0,C 180,E1 -23048.884,E2 -23048.884} C_VEL
LIN {X 0,Y 226.578,Z 755.139,A -85,B 0,C 180,E1 -23052.005,E2 -23052.005} C_VEL
LIN {X 0,Y 227.952,Z 756.688,A -85,B 0,C 180,E1 -23053.711,E2 -23053.711} C_VEL
LIN {X 0,Y 230.74,Z 760.748,A -85,B 0,C 180,E1 -23056.706,E2 -23056.706} C_VEL
LIN {X 0,Y 234.264,Z 766.033,A -85,B 0,C 180,E1 -23059.811,E2 -23059.811} C_VEL
LIN {X 0,Y 237.398,Z 770.909,A -85,B 0,C 180,E1 -23062.176,E2 -23062.176} C_VEL
LIN {X 0,Y 241.506,Z 777.633,A -85,B 0,C 180,E1 -23064.901,E2 -23064.901} C_VEL
LIN {X 0,Y 245.746,Z 786.859,A -85,B 0,C 180,E1 -23067.508,E2 -23067.508} C_VEL
LIN {X 0,Y 249.579,Z 795.951,A -85,B 0,C 180,E1 -23069.658,E2 -23069.658} C_VEL
LIN {X 0,Y 251.673,Z 801.402,A -85,B 0,C 180,E1 -23070.776,E2 -23070.776} C_VEL
LIN {X 0,Y 244.555,Z 888.594,A -85,B 0,C 180,E1 -23072.902,E2 -23072.902} C_VEL
LIN {X 0,Y 242.665,Z 902.347,A -85,B 0,C 180,E1 -23073.378,E2 -23073.378} C_VEL
LIN {X 0,Y 240.262,Z 914.83,A -85,B 0,C 180,E1 -23073.923,E2 -23073.923} C_VEL
LIN {X 0,Y 237.362,Z 926.738,A -85,B 0,C 180,E1 -23074.566,E2 -23074.566} C_VEL
LIN {X 0,Y 234.525,Z 936.922,A -85,B 0,C 180,E1 -23075.256,E2 -23075.256} C_VEL
LIN {X 0,Y 230.25,Z 950.152,A -85,B 0,C 180,E1 -23076.387,E2 -23076.387} C_VEL
LIN {X 0,Y 225.452,Z 962.881,A -85,B 0,C 180,E1 -23077.722,E2 -23077.722} C_VEL
LIN {X 0,Y 220.796,Z 973.87,A -85,B 0,C 180,E1 -23079.119,E2 -23079.119} C_VEL
LIN {X 0,Y 215.795,Z 984.601,A -85,B 0,C 180,E1 -23080.763,E2 -23080.763} C_VEL
LIN {X 0,Y 210.363,Z 995.155,A -85,B 0,C 180,E1 -23082.695,E2 -23082.695} C_VEL
LIN {X 0,Y 205.204,Z 1004.417,A -85,B 0,C 180,E1 -23084.713,E2 -23084.713} C_VEL
LIN {X 0,Y 199.453,Z 1014.145,A -85,B 0,C 180,E1 -23087.29,E2 -23087.29} C_VEL
LIN {X 0,Y 193.319,Z 1023.947,A -85,B 0,C 180,E1 -23090.492,E2 -23090.492} C_VEL
LIN {X 0,Y 188.473,Z 1031.265,A -85,B 0,C 180,E1 -23093.372,E2 -23093.372} C_VEL
LIN {X 0,Y 184.198,Z 1037.697,A -85,B 0,C 180,E1 -23096.411,E2 -23096.411} C_VEL
LIN {X 0,Y 179.814,Z 1044.194,A -85,B 0,C 180,E1 -23100.145,E2 -23100.145} C_VEL
LIN {X 0,Y 177.563,Z 1046.684,A -85,B 0,C 180,E1 -23101.718,E2 -23101.718} C_VEL
LIN {X 0,Y 172.401,Z 1050.399,A -85,B 0,C 180,E1 -23104.21,E2 -23104.21} C_VEL
LIN {X 0,Y 167.488,Z 1053.779,A -85,B 0,C 180,E1 -23106.891,E2 -23106.891} C_VEL
LIN {X 0,Y 165.683,Z 1055.491,A -85,B 0,C 180,E1 -23108.724,E2 -23108.724} C_VEL
LIN {X 0,Y 163.001,Z 1060.214,A -85,B 0,C 180,E1 -23115.008,E2 -23115.008} C_VEL
LIN {X 0,Y 161.973,Z 1062.7,A -85,B 0,C 180,E1 -23120.005,E2 -23120.005} C_VEL
LIN {X 0,Y 161.69,Z 1064.188,A -85,B 0,C 180,E1 -23125.013,E2 -23125.013} C_VEL
LIN {X 0,Y 161.896,Z 1064.689,A -85,B 0,C 180,E1 -23130,E2 -23130} C_VEL
LIN {X 0,Y 161.69,Z 1064.188,A -85,B 0,C 180,E1 -23134.987,E2 -23134.987} C_VEL
LIN {X 0,Y 161.973,Z 1062.7,A -85,B 0,C 180,E1 -23139.995,E2 -23139.995} C_VEL
LIN {X 0,Y 163.001,Z 1060.214,A -85,B 0,C 180,E1 -23144.992,E2 -23144.992} C_VEL
LIN {X 0,Y 165.441,Z 1055.883,A -85,B 0,C 180,E1 -23150.841,E2 -23150.841} C_VEL
LIN {X 0,Y 167.92,Z 1052.113,A -85,B 0,C 180,E1 -23154.741,E2 -23154.741} C_VEL
LIN {X 0,Y 171.89,Z 1046.378,A -85,B 0,C 180,E1 -23159.382,E2 -23159.382} C_VEL
LIN {X 0,Y 175.483,Z 1041.282,A -85,B 0,C 180,E1 -23162.749,E2 -23162.749} C_VEL
LIN {X 0,Y 181.206,Z 1033.28,A -85,B 0,C 180,E1 -23166.952,E2 -23166.952} C_VEL
LIN {X 0,Y 186.146,Z 1026.3,A -85,B 0,C 180,E1 -23169.928,E2 -23169.928} C_VEL
LIN {X 0,Y 191.235,Z 1018.623,A -85,B 0,C 180,E1 -23172.691,E2 -23172.691} C_VEL
LIN {X 0,Y 197.192,Z 1009.224,A -85,B 0,C 180,E1 -23175.462,E2 -23175.462} C_VEL
LIN {X 0,Y 202.268,Z 1000.658,A -85,B 0,C 180,E1 -23177.589,E2 -23177.589} C_VEL
LIN {X 0,Y 208.904,Z 988.806,A -85,B 0,C 180,E1 -23179.937,E2 -23179.937} C_VEL
LIN {X 0,Y 214.118,Z 978.454,A -85,B 0,C 180,E1 -23181.653,E2 -23181.653} C_VEL
LIN {X 0,Y 219.336,Z 966.986,A -85,B 0,C 180,E1 -23183.229,E2 -23183.229} C_VEL
LIN {X 0,Y 224.235,Z 954.969,A -85,B 0,C 180,E1 -23184.575,E2 -23184.575} C_VEL
LIN {X 0,Y 228.593,Z 942.657,A -85,B 0,C 180,E1 -23185.714,E2 -23185.714} C_VEL
LIN {X 0,Y 232.41,Z 930.119,A -85,B 0,C 180,E1 -23186.652,E2 -23186.652} C_VEL
LIN {X 0,Y 235.944,Z 916.4,A -85,B 0,C 180,E1 -23187.432,E2 -23187.432} C_VEL
LIN {X 0,Y 238.598,Z 903.51,A -85,B 0,C 180,E1 -23187.995,E2 -23187.995} C_VEL
LIN {X 0,Y 240.569,Z 890.106,A -85,B 0,C 180,E1 -23188.463,E2 -23188.463} C_VEL
LIN {X 0,Y 243.043,Z 862.373,A -85,B 0,C 180,E1 -23189.184,E2 -23189.184} C_VEL
LIN {X 0,Y 247.795,Z 804.159,A -85,B 0,C 180,E1 -23190.593,E2 -23190.593} C_VEL
LIN {X 0,Y 243.859,Z 794.108,A -85,B 0,C 180,E1 -23192.889,E2 -23192.889} C_VEL
LIN {X 0,Y 239.803,Z 784.809,A -85,B 0,C 180,E1 -23195.473,E2 -23195.473} C_VEL
LIN {X 0,Y 238.196,Z 781.707,A -85,B 0,C 180,E1 -23196.554,E2 -23196.554} C_VEL
LIN {X 0,Y 233.894,Z 774.575,A -85,B 0,C 180,E1 -23199.693,E2 -23199.693} C_VEL
LIN {X 0,Y 231.286,Z 770.625,A -85,B 0,C 180,E1 -23201.874,E2 -23201.874} C_VEL
LIN {X 0,Y 228.995,Z 767.083,A -85,B 0,C 180,E1 -23204.079,E2 -23204.079} C_VEL
LIN {X 0,Y 226.285,Z 762.94,A -85,B 0,C 180,E1 -23207.215,E2 -23207.215} C_VEL
LIN {X 0,Y 223.959,Z 759.53,A -85,B 0,C 180,E1 -23210.745,E2 -23210.745} C_VEL
LIN {X 0,Y 223.422,Z 758.355,A -85,B 0,C 180,E1 -23211.862,E2 -23211.862} C_VEL
LIN {X 0,Y 221.425,Z 755.382,A -85,B 0,C 180,E1 -23220,E2 -23220} C_VEL
LIN {X 0,Y 223.627,Z 758.638,A -85,B 0,C 180,E1 -23228.955,E2 -23228.955} C_VEL
LIN {X 0,Y 225.641,Z 762.271,A -85,B 0,C 180,E1 -23232.364,E2 -23232.364} C_VEL
LIN {X 0,Y 226.801,Z 763.633,A -85,B 0,C 180,E1 -23233.838,E2 -23233.838} C_VEL
LIN {X 0,Y 229.999,Z 768.651,A -85,B 0,C 180,E1 -23237.335,E2 -23237.335} C_VEL
LIN {X 0,Y 232.761,Z 772.84,A -85,B 0,C 180,E1 -23239.799,E2 -23239.799} C_VEL
LIN {X 0,Y 236.637,Z 779.023,A -85,B 0,C 180,E1 -23242.769,E2 -23242.769} C_VEL
LIN {X 0,Y 241.868,Z 787.981,A -85,B 0,C 180,E1 -23246.187,E2 -23246.187} C_VEL
LIN {X 0,Y 251.91,Z 804.523,A -85,B 0,C 180,E1 -23251.441,E2 -23251.441} C_VEL
LIN {X 0,Y 259.367,Z 813.786,A -85,B 0,C 180,E1 -23254.508,E2 -23254.508} C_VEL
LIN {X 0,Y 267.012,Z 821.816,A -85,B 0,C 180,E1 -23257.196,E2 -23257.196} C_VEL
LIN {X 0,Y 283.454,Z 835.979,A -85,B 0,C 180,E1 -23261.951,E2 -23261.951} C_VEL
LIN {X 0,Y 291.365,Z 842.288,A -85,B 0,C 180,E1 -23264.145,E2 -23264.145} C_VEL
LIN {X 0,Y 297.23,Z 846.98,A -85,B 0,C 180,E1 -23265.891,E2 -23265.891} C_VEL
LIN {X 0,Y 302.646,Z 851.387,A -85,B 0,C 180,E1 -23267.617,E2 -23267.617} C_VEL
LIN {X 0,Y 307.44,Z 855.375,A -85,B 0,C 180,E1 -23269.257,E2 -23269.257} C_VEL
LIN {X 0,Y 313.851,Z 860.486,A -85,B 0,C 180,E1 -23271.604,E2 -23271.604} C_VEL
LIN {X 0,Y 320.827,Z 866.371,A -85,B 0,C 180,E1 -23274.347,E2 -23274.347} C_VEL
LIN {X 0,Y 325.654,Z 870.287,A -85,B 0,C 180,E1 -23276.326,E2 -23276.326} C_VEL
LIN {X 0,Y 331.354,Z 874.898,A -85,B 0,C 180,E1 -23278.789,E2 -23278.789} C_VEL
LIN {X 0,Y 334.978,Z 877.659,A -85,B 0,C 180,E1 -23280.419,E2 -23280.419} C_VEL
LIN {X 0,Y 339.292,Z 881.251,A -85,B 0,C 180,E1 -23282.495,E2 -23282.495} C_VEL
LIN {X 0,Y 344.24,Z 884.61,A -85,B 0,C 180,E1 -23284.997,E2 -23284.997} C_VEL
LIN {X 0,Y 348.516,Z 888.282,A -85,B 0,C 180,E1 -23287.399,E2 -23287.399} C_VEL
LIN {X 0,Y 352.663,Z 891.223,A -85,B 0,C 180,E1 -23289.918,E2 -23289.918} C_VEL
LIN {X 0,Y 356.24,Z 893.508,A -85,B 0,C 180,E1 -23292.358,E2 -23292.358} C_VEL
LIN {X 0,Y 359.465,Z 896.454,A -85,B 0,C 180,E1 -23294.952,E2 -23294.952} C_VEL
LIN {X 0,Y 362.241,Z 898.447,A -85,B 0,C 180,E1 -23297.498,E2 -23297.498} C_VEL
LIN {X 0,Y 364.514,Z 899.741,A -85,B 0,C 180,E1 -23300.007,E2 -23300.007} C_VEL
LIN {X 0,Y 366.153,Z 900.505,A -85,B 0,C 180,E1 -23302.279,E2 -23302.279} C_VEL
LIN {X 0,Y 367.352,Z 901.04,A -85,B 0,C 180,E1 -23304.511,E2 -23304.511} C_VEL
LIN {X 0,Y 368.19,Z 901.456,A -85,B 0,C 180,E1 -23306.717,E2 -23306.717} C_VEL
LIN {X 0,Y 368.632,Z 901.689,A -85,B 0,C 180,E1 -23310,E2 -23310} C_VEL
LIN {X 0,Y 368.19,Z 901.457,A -85,B 0,C 180,E1 -23313.283,E2 -23313.283} C_VEL
LIN {X 0,Y 367.258,Z 900.986,A -85,B 0,C 180,E1 -23315.686,E2 -23315.686} C_VEL
LIN {X 0,Y 365.987,Z 900.41,A -85,B 0,C 180,E1 -23318.028,E2 -23318.028} C_VEL
LIN {X 0,Y 364.046,Z 899.503,A -85,B 0,C 180,E1 -23320.527,E2 -23320.527} C_VEL
LIN {X 0,Y 361.646,Z 898.087,A -85,B 0,C 180,E1 -23323.087,E2 -23323.087} C_VEL
LIN {X 0,Y 358.863,Z 895.911,A -85,B 0,C 180,E1 -23325.58,E2 -23325.58} C_VEL
LIN {X 0,Y 355.319,Z 892.763,A -85,B 0,C 180,E1 -23328.305,E2 -23328.305} C_VEL
LIN {X 0,Y 351.451,Z 890.452,A -85,B 0,C 180,E1 -23330.824,E2 -23330.824} C_VEL
LIN {X 0,Y 347.24,Z 887.197,A -85,B 0,C 180,E1 -23333.339,E2 -23333.339} C_VEL
LIN {X 0,Y 343.404,Z 884.037,A -85,B 0,C 180,E1 -23335.453,E2 -23335.453} C_VEL
LIN {X 0,Y 338.263,Z 880.505,A -85,B 0,C 180,E1 -23338.014,E2 -23338.014} C_VEL
LIN {X 0,Y 332.569,Z 875.685,A -85,B 0,C 180,E1 -23340.688,E2 -23340.688} C_VEL
LIN {X 0,Y 327.249,Z 871.674,A -85,B 0,C 180,E1 -23343,E2 -23343} C_VEL
LIN {X 0,Y 321.803,Z 867.089,A -85,B 0,C 180,E1 -23345.264,E2 -23345.264} C_VEL
LIN {X 0,Y 315.487,Z 861.87,A -85,B 0,C 180,E1 -23347.764,E2 -23347.764} C_VEL
LIN {X 0,Y 308.862,Z 856.602,A -85,B 0,C 180,E1 -23350.221,E2 -23350.221} C_VEL
LIN {X 0,Y 303.219,Z 851.812,A -85,B 0,C 180,E1 -23352.193,E2 -23352.193} C_VEL
LIN {X 0,Y 297.706,Z 847.382,A -85,B 0,C 180,E1 -23353.957,E2 -23353.957} C_VEL
LIN {X 0,Y 291.87,Z 842.666,A -85,B 0,C 180,E1 -23355.71,E2 -23355.71} C_VEL
LIN {X 0,Y 283.922,Z 836.338,A -85,B 0,C 180,E1 -23357.922,E2 -23357.922} C_VEL
LIN {X 0,Y 269.001,Z 823.634,A -85,B 0,C 180,E1 -23362.167,E2 -23362.167} C_VEL
LIN {X 0,Y 260.577,Z 815.194,A -85,B 0,C 180,E1 -23365.038,E2 -23365.038} C_VEL
LIN {X 0,Y 251.392,Z 803.836,A -85,B 0,C 180,E1 -23368.791,E2 -23368.791} C_VEL
LIN {X 0,Y 240.016,Z 784.775,A -85,B 0,C 180,E1 -23374.959,E2 -23374.959} C_VEL
LIN {X 0,Y 235.372,Z 777.067,A -85,B 0,C 180,E1 -23378.142,E2 -23378.142} C_VEL
LIN {X 0,Y 231.759,Z 771.221,A -85,B 0,C 180,E1 -23381.061,E2 -23381.061} C_VEL
LIN {X 0,Y 228.936,Z 767.01,A -85,B 0,C 180,E1 -23383.732,E2 -23383.732} C_VEL
LIN {X 0,Y 226.328,Z 762.928,A -85,B 0,C 180,E1 -23386.762,E2 -23386.762} C_VEL
LIN {X 0,Y 224.16,Z 759.966,A -85,B 0,C 180,E1 -23389.953,E2 -23389.953} C_VEL
LIN {X 0,Y 223.446,Z 758.377,A -85,B 0,C 180,E1 -23391.408,E2 -23391.408} C_VEL
LIN {X 0,Y 221.425,Z 755.383,A -85,B 0,C 180,E1 -23400,E2 -23400} C_VEL
LIN {X 0,Y 223.646,Z 758.663,A -85,B 0,C 180,E1 -23408.585,E2 -23408.585} C_VEL
LIN {X 0,Y 225.484,Z 762.08,A -85,B 0,C 180,E1 -23411.743,E2 -23411.743} C_VEL
LIN {X 0,Y 226.712,Z 763.584,A -85,B 0,C 180,E1 -23413.33,E2 -23413.33} C_VEL
LIN {X 0,Y 229.841,Z 768.4,A -85,B 0,C 180,E1 -23416.773,E2 -23416.773} C_VEL
LIN {X 0,Y 232.705,Z 772.759,A -85,B 0,C 180,E1 -23419.346,E2 -23419.346} C_VEL
LIN {X 0,Y 235.932,Z 777.947,A -85,B 0,C 180,E1 -23421.861,E2 -23421.861} C_VEL
LIN {X 0,Y 239.273,Z 783.638,A -85,B 0,C 180,E1 -23424.166,E2 -23424.166} C_VEL
LIN {X 0,Y 243.701,Z 793.71,A -85,B 0,C 180,E1 -23427.014,E2 -23427.014} C_VEL
LIN {X 0,Y 247.837,Z 804.26,A -85,B 0,C 180,E1 -23429.43,E2 -23429.43} C_VEL
LIN {X 0,Y 240.843,Z 887.677,A -85,B 0,C 180,E1 -23431.457,E2 -23431.457} C_VEL
LIN {X 0,Y 238.925,Z 901.541,A -85,B 0,C 180,E1 -23431.93,E2 -23431.93} C_VEL
LIN {X 0,Y 236.591,Z 913.529,A -85,B 0,C 180,E1 -23432.432,E2 -23432.432} C_VEL
LIN {X 0,Y 233.409,Z 926.533,A -85,B 0,C 180,E1 -23433.132,E2 -23433.132} C_VEL
LIN {X 0,Y 230.485,Z 936.716,A -85,B 0,C 180,E1 -23433.81,E2 -23433.81} C_VEL
LIN {X 0,Y 226.097,Z 949.945,A -85,B 0,C 180,E1 -23434.933,E2 -23434.933} C_VEL
LIN {X 0,Y 221.168,Z 962.675,A -85,B 0,C 180,E1 -23436.263,E2 -23436.263} C_VEL
LIN {X 0,Y 216.346,Z 973.662,A -85,B 0,C 180,E1 -23437.646,E2 -23437.646} C_VEL
LIN {X 0,Y 210.753,Z 985.227,A -85,B 0,C 180,E1 -23439.435,E2 -23439.435} C_VEL
LIN {X 0,Y 205.582,Z 994.948,A -85,B 0,C 180,E1 -23441.23,E2 -23441.23} C_VEL
LIN {X 0,Y 200.218,Z 1004.209,A -85,B 0,C 180,E1 -23443.252,E2 -23443.252} C_VEL
LIN {X 0,Y 194.22,Z 1013.937,A -85,B 0,C 180,E1 -23445.849,E2 -23445.849} C_VEL
LIN {X 0,Y 188.677,Z 1022.459,A -85,B 0,C 180,E1 -23448.612,E2 -23448.612} C_VEL
LIN {X 0,Y 182.731,Z 1031.056,A -85,B 0,C 180,E1 -23452.022,E2 -23452.022} C_VEL
LIN {X 0,Y 178.221,Z 1037.488,A -85,B 0,C 180,E1 -23455.125,E2 -23455.125} C_VEL
LIN {X 0,Y 173.018,Z 1044.754,A -85,B 0,C 180,E1 -23459.487,E2 -23459.487} C_VEL
LIN {X 0,Y 169.751,Z 1049.41,A -85,B 0,C 180,E1 -23462.909,E2 -23462.909} C_VEL
LIN {X 0,Y 166.326,Z 1054.519,A -85,B 0,C 180,E1 -23467.649,E2 -23467.649} C_VEL
LIN {X 0,Y 165.683,Z 1055.491,A -85,B 0,C 180,E1 -23468.724,E2 -23468.724} C_VEL
LIN {X 0,Y 164.013,Z 1057.225,A -85,B 0,C 180,E1 -23470.61,E2 -23470.61} C_VEL
LIN {X 0,Y 159.822,Z 1059.457,A -85,B 0,C 180,E1 -23473.687,E2 -23473.687} C_VEL
LIN {X 0,Y 156.621,Z 1060.983,A -85,B 0,C 180,E1 -23476.272,E2 -23476.272} C_VEL
LIN {X 0,Y 155.169,Z 1061.953,A -85,B 0,C 180,E1 -23478.352,E2 -23478.352} C_VEL
LIN {X 0,Y 154.985,Z 1062.275,A -85,B 0,C 180,E1 -23479.068,E2 -23479.068} C_VEL
LIN {X 0,Y 154.607,Z 1063.982,A -85,B 0,C 180,E1 -23484.784,E2 -23484.784} C_VEL
LIN {X 0,Y 154.794,Z 1064.484,A -85,B 0,C 180,E1 -23490,E2 -23490} C_VEL
LIN {X 0,Y 154.607,Z 1063.982,A -85,B 0,C 180,E1 -23495.216,E2 -23495.216} C_VEL
LIN {X 0,Y 154.93,Z 1062.493,A -85,B 0,C 180,E1 -23500.454,E2 -23500.454} C_VEL
LIN {X 0,Y 156.093,Z 1060.006,A -85,B 0,C 180,E1 -23505.673,E2 -23505.673} C_VEL
LIN {X 0,Y 158.543,Z 1055.969,A -85,B 0,C 180,E1 -23511.424,E2 -23511.424} C_VEL
LIN {X 0,Y 161.398,Z 1051.904,A -85,B 0,C 180,E1 -23515.813,E2 -23515.813} C_VEL
LIN {X 0,Y 165.642,Z 1046.169,A -85,B 0,C 180,E1 -23520.606,E2 -23520.606} C_VEL
LIN {X 0,Y 169.731,Z 1040.722,A -85,B 0,C 180,E1 -23524.271,E2 -23524.271} C_VEL
LIN {X 0,Y 175.484,Z 1033.071,A -85,B 0,C 180,E1 -23528.371,E2 -23528.371} C_VEL
LIN {X 0,Y 180.678,Z 1026.092,A -85,B 0,C 180,E1 -23531.395,E2 -23531.395} C_VEL
LIN {X 0,Y 186.458,Z 1017.71,A -85,B 0,C 180,E1 -23534.422,E2 -23534.422} C_VEL
LIN {X 0,Y 192.215,Z 1009.016,A -85,B 0,C 180,E1 -23536.991,E2 -23536.991} C_VEL
LIN {X 0,Y 197.512,Z 1000.451,A -85,B 0,C 180,E1 -23539.123,E2 -23539.123} C_VEL
LIN {X 0,Y 204.369,Z 988.599,A -85,B 0,C 180,E1 -23541.474,E2 -23541.474} C_VEL
LIN {X 0,Y 209.692,Z 978.369,A -85,B 0,C 180,E1 -23543.169,E2 -23543.169} C_VEL
LIN {X 0,Y 215.133,Z 966.779,A -85,B 0,C 180,E1 -23544.754,E2 -23544.754} C_VEL
LIN {X 0,Y 220.186,Z 954.763,A -85,B 0,C 180,E1 -23546.084,E2 -23546.084} C_VEL
LIN {X 0,Y 224.659,Z 942.451,A -85,B 0,C 180,E1 -23547.215,E2 -23547.215} C_VEL
LIN {X 0,Y 228.581,Z 929.914,A -85,B 0,C 180,E1 -23548.14,E2 -23548.14} C_VEL
LIN {X 0,Y 232.209,Z 916.129,A -85,B 0,C 180,E1 -23548.914,E2 -23548.914} C_VEL
LIN {X 0,Y 234.877,Z 903.495,A -85,B 0,C 180,E1 -23549.458,E2 -23549.458} C_VEL
LIN {X 0,Y 236.872,Z 890.377,A -85,B 0,C 180,E1 -23549.916,E2 -23549.916} C_VEL
LIN {X 0,Y 239.277,Z 864.595,A -85,B 0,C 180,E1 -23550.586,E2 -23550.586} C_VEL
LIN {X 0,Y 244.14,Z 807.274,A -85,B 0,C 180,E1 -23551.949,E2 -23551.949} C_VEL
LIN {X 0,Y 240.442,Z 797.6,A -85,B 0,C 180,E1 -23554.275,E2 -23554.275} C_VEL
LIN {X 0,Y 236.647,Z 788.662,A -85,B 0,C 180,E1 -23556.897,E2 -23556.897} C_VEL
LIN {X 0,Y 232,Z 780.767,A -85,B 0,C 180,E1 -23560.42,E2 -23560.42} C_VEL
LIN {X 0,Y 229.386,Z 776.701,A -85,B 0,C 180,E1 -23562.734,E2 -23562.734} C_VEL
LIN {X 0,Y 227.499,Z 773.652,A -85,B 0,C 180,E1 -23564.661,E2 -23564.661} C_VEL
LIN {X 0,Y 225.077,Z 769.772,A -85,B 0,C 180,E1 -23567.603,E2 -23567.603} C_VEL
LIN {X 0,Y 222.795,Z 766.232,A -85,B 0,C 180,E1 -23571.268,E2 -23571.268} C_VEL
LIN {X 0,Y 222.334,Z 765.261,A -85,B 0,C 180,E1 -23572.279,E2 -23572.279} C_VEL
LIN {X 0,Y 220.559,Z 762.435,A -85,B 0,C 180,E1 -23580,E2 -23580} C_VEL
LIN {X 0,Y 222.585,Z 765.605,A -85,B 0,C 180,E1 -23588.654,E2 -23588.654} C_VEL
LIN {X 0,Y 224.496,Z 769.151,A -85,B 0,C 180,E1 -23592.027,E2 -23592.027} C_VEL
LIN {X 0,Y 225.528,Z 770.465,A -85,B 0,C 180,E1 -23593.401,E2 -23593.401} C_VEL
LIN {X 0,Y 228.501,Z 775.252,A -85,B 0,C 180,E1 -23596.798,E2 -23596.798} C_VEL
LIN {X 0,Y 231.129,Z 779.406,A -85,B 0,C 180,E1 -23599.252,E2 -23599.252} C_VEL
LIN {X 0,Y 234.547,Z 785.043,A -85,B 0,C 180,E1 -23601.998,E2 -23601.998} C_VEL
LIN {X 0,Y 239.642,Z 794.067,A -85,B 0,C 180,E1 -23605.494,E2 -23605.494} C_VEL
LIN {X 0,Y 249.146,Z 810.212,A -85,B 0,C 180,E1 -23610.695,E2 -23610.695} C_VEL
LIN {X 0,Y 256.72,Z 819.854,A -85,B 0,C 180,E1 -23613.932,E2 -23613.932} C_VEL
LIN {X 0,Y 264.43,Z 828.039,A -85,B 0,C 180,E1 -23616.726,E2 -23616.726} C_VEL
LIN {X 0,Y 280.218,Z 841.853,A -85,B 0,C 180,E1 -23621.414,E2 -23621.414} C_VEL
LIN {X 0,Y 289.036,Z 848.775,A -85,B 0,C 180,E1 -23623.806,E2 -23623.806} C_VEL
LIN {X 0,Y 295.948,Z 854.291,A -85,B 0,C 180,E1 -23625.845,E2 -23625.845} C_VEL
LIN {X 0,Y 301.818,Z 858.883,A -85,B 0,C 180,E1 -23627.702,E2 -23627.702} C_VEL
LIN {X 0,Y 307.412,Z 863.577,A -85,B 0,C 180,E1 -23629.631,E2 -23629.631} C_VEL
LIN {X 0,Y 313.83,Z 868.67,A -85,B 0,C 180,E1 -23631.991,E2 -23631.991} C_VEL
LIN {X 0,Y 319.906,Z 873.649,A -85,B 0,C 180,E1 -23634.374,E2 -23634.374} C_VEL
LIN {X 0,Y 325.179,Z 878.032,A -85,B 0,C 180,E1 -23636.545,E2 -23636.545} C_VEL
LIN {X 0,Y 330.775,Z 882.317,A -85,B 0,C 180,E1 -23638.954,E2 -23638.954} C_VEL
LIN {X 0,Y 336.886,Z 887.346,A -85,B 0,C 180,E1 -23641.778,E2 -23641.778} C_VEL
LIN {X 0,Y 341.974,Z 890.929,A -85,B 0,C 180,E1 -23644.295,E2 -23644.295} C_VEL
LIN {X 0,Y 344.23,Z 892.62,A -85,B 0,C 180,E1 -23645.493,E2 -23645.493} C_VEL
LIN {X 0,Y 348.273,Z 895.921,A -85,B 0,C 180,E1 -23647.801,E2 -23647.801} C_VEL
LIN {X 0,Y 352.34,Z 898.709,A -85,B 0,C 180,E1 -23650.311,E2 -23650.311} C_VEL
LIN {X 0,Y 355.159,Z 900.49,A -85,B 0,C 180,E1 -23652.232,E2 -23652.232} C_VEL
LIN {X 0,Y 358.321,Z 903.349,A -85,B 0,C 180,E1 -23654.734,E2 -23654.734} C_VEL
LIN {X 0,Y 361.156,Z 905.379,A -85,B 0,C 180,E1 -23657.27,E2 -23657.27} C_VEL
LIN {X 0,Y 363.387,Z 906.687,A -85,B 0,C 180,E1 -23659.728,E2 -23659.728} C_VEL
LIN {X 0,Y 365.273,Z 907.549,A -85,B 0,C 180,E1 -23662.26,E2 -23662.26} C_VEL
LIN {X 0,Y 366.477,Z 908.081,A -85,B 0,C 180,E1 -23664.498,E2 -23664.498} C_VEL
LIN {X 0,Y 367.323,Z 908.501,A -85,B 0,C 180,E1 -23666.71,E2 -23666.71} C_VEL
LIN {X 0,Y 367.675,Z 908.675,A -85,B 0,C 180,E1 -23668.905,E2 -23668.905} C_VEL
LIN {X 0,Y 367.675,Z 908.675,A -85,B 0,C 180,E1 -23671.095,E2 -23671.095} C_VEL
LIN {X 0,Y 367.323,Z 908.503,A -85,B 0,C 180,E1 -23673.29,E2 -23673.29} C_VEL
LIN {X 0,Y 366.476,Z 908.094,A -85,B 0,C 180,E1 -23675.502,E2 -23675.502} C_VEL
LIN {X 0,Y 365.273,Z 907.546,A -85,B 0,C 180,E1 -23677.74,E2 -23677.74} C_VEL
LIN {X 0,Y 363.262,Z 906.614,A -85,B 0,C 180,E1 -23680.418,E2 -23680.418} C_VEL
LIN {X 0,Y 360.943,Z 905.25,A -85,B 0,C 180,E1 -23682.929,E2 -23682.929} C_VEL
LIN {X 0,Y 358.125,Z 903.144,A -85,B 0,C 180,E1 -23685.443,E2 -23685.443} C_VEL
LIN {X 0,Y 354.951,Z 900.269,A -85,B 0,C 180,E1 -23687.921,E2 -23687.921} C_VEL
LIN {X 0,Y 350.927,Z 897.781,A -85,B 0,C 180,E1 -23690.59,E2 -23690.59} C_VEL
LIN {X 0,Y 346.695,Z 894.664,A -85,B 0,C 180,E1 -23693.129,E2 -23693.129} C_VEL
LIN {X 0,Y 342.085,Z 890.916,A -85,B 0,C 180,E1 -23695.655,E2 -23695.655} C_VEL
LIN {X 0,Y 336.883,Z 887.367,A -85,B 0,C 180,E1 -23698.222,E2 -23698.222} C_VEL
LIN {X 0,Y 331.125,Z 882.541,A -85,B 0,C 180,E1 -23700.894,E2 -23700.894} C_VEL
LIN {X 0,Y 325.586,Z 878.386,A -85,B 0,C 180,E1 -23703.282,E2 -23703.282} C_VEL
LIN {X 0,Y 319.54,Z 873.366,A -85,B 0,C 180,E1 -23705.775,E2 -23705.775} C_VEL
LIN {X 0,Y 313.218,Z 868.09,A -85,B 0,C 180,E1 -23708.25,E2 -23708.25} C_VEL
LIN {X 0,Y 306.786,Z 863.069,A -85,B 0,C 180,E1 -23710.595,E2 -23710.595} C_VEL
LIN {X 0,Y 299.48,Z 857.037,A -85,B 0,C 180,E1 -23713.078,E2 -23713.078} C_VEL
LIN {X 0,Y 291.652,Z 850.804,A -85,B 0,C 180,E1 -23715.438,E2 -23715.438} C_VEL
LIN {X 0,Y 284.74,Z 845.317,A -85,B 0,C 180,E1 -23717.374,E2 -23717.374} C_VEL
LIN {X 0,Y 268.806,Z 832.248,A -85,B 0,C 180,E1 -23721.853,E2 -23721.853} C_VEL
LIN {X 0,Y 257.627,Z 820.904,A -85,B 0,C 180,E1 -23725.715,E2 -23725.715} C_VEL
LIN {X 0,Y 249.7,Z 810.974,A -85,B 0,C 180,E1 -23729.048,E2 -23729.048} C_VEL
LIN {X 0,Y 241.968,Z 798.505,A -85,B 0,C 180,E1 -23733.076,E2 -23733.076} C_VEL
LIN {X 0,Y 237.63,Z 790.451,A -85,B 0,C 180,E1 -23735.815,E2 -23735.815} C_VEL
LIN {X 0,Y 233.227,Z 782.886,A -85,B 0,C 180,E1 -23739.01,E2 -23739.01} C_VEL
LIN {X 0,Y 229.897,Z 777.419,A -85,B 0,C 180,E1 -23741.855,E2 -23741.855} C_VEL
LIN {X 0,Y 227.444,Z 773.564,A -85,B 0,C 180,E1 -23744.314,E2 -23744.314} C_VEL
LIN {X 0,Y 225.121,Z 769.755,A -85,B 0,C 180,E1 -23747.149,E2 -23747.149} C_VEL
LIN {X 0,Y 223.048,Z 766.808,A -85,B 0,C 180,E1 -23750.346,E2 -23750.346} C_VEL
LIN {X 0,Y 222.356,Z 765.292,A -85,B 0,C 180,E1 -23751.824,E2 -23751.824} C_VEL
LIN {X 0,Y 220.559,Z 762.436,A -85,B 0,C 180,E1 -23760,E2 -23760} C_VEL
LIN {X 0,Y 222.601,Z 765.636,A -85,B 0,C 180,E1 -23768.283,E2 -23768.283} C_VEL
LIN {X 0,Y 224.399,Z 768.993,A -85,B 0,C 180,E1 -23771.477,E2 -23771.477} C_VEL
LIN {X 0,Y 225.485,Z 770.457,A -85,B 0,C 180,E1 -23772.946,E2 -23772.946} C_VEL
LIN {X 0,Y 228.522,Z 775.29,A -85,B 0,C 180,E1 -23776.413,E2 -23776.413} C_VEL
LIN {X 0,Y 231.249,Z 779.597,A -85,B 0,C 180,E1 -23778.948,E2 -23778.948} C_VEL
LIN {X 0,Y 234.65,Z 785.228,A -85,B 0,C 180,E1 -23781.669,E2 -23781.669} C_VEL
LIN {X 0,Y 237.054,Z 789.634,A -85,B 0,C 180,E1 -23783.402,E2 -23783.402} C_VEL
LIN {X 0,Y 241.058,Z 799.099,A -85,B 0,C 180,E1 -23786.123,E2 -23786.123} C_VEL
LIN {X 0,Y 244.102,Z 807.152,A -85,B 0,C 180,E1 -23788.027,E2 -23788.027} C_VEL
LIN {X 0,Y 241.672,Z 836.285,A -85,B 0,C 180,E1 -23788.739,E2 -23788.739} C_VEL
LIN {X 0,Y 237.144,Z 888.091,A -85,B 0,C 180,E1 -23790.013,E2 -23790.013} C_VEL
LIN {X 0,Y 235.243,Z 901.318,A -85,B 0,C 180,E1 -23790.459,E2 -23790.459} C_VEL
LIN {X 0,Y 232.741,Z 913.864,A -85,B 0,C 180,E1 -23790.984,E2 -23790.984} C_VEL
LIN {X 0,Y 229.609,Z 926.328,A -85,B 0,C 180,E1 -23791.649,E2 -23791.649} C_VEL
LIN {X 0,Y 226.599,Z 936.51,A -85,B 0,C 180,E1 -23792.313,E2 -23792.313} C_VEL
LIN {X 0,Y 222.105,Z 949.74,A -85,B 0,C 180,E1 -23793.431,E2 -23793.431} C_VEL
LIN {X 0,Y 217.013,Z 962.468,A -85,B 0,C 180,E1 -23794.74,E2 -23794.74} C_VEL
LIN {X 0,Y 212.052,Z 973.456,A -85,B 0,C 180,E1 -23796.115,E2 -23796.115} C_VEL
LIN {X 0,Y 206.733,Z 984.109,A -85,B 0,C 180,E1 -23797.729,E2 -23797.729} C_VEL
LIN {X 0,Y 200.947,Z 994.741,A -85,B 0,C 180,E1 -23799.699,E2 -23799.699} C_VEL
LIN {X 0,Y 195.377,Z 1004.002,A -85,B 0,C 180,E1 -23801.722,E2 -23801.722} C_VEL
LIN {X 0,Y 189.124,Z 1013.729,A -85,B 0,C 180,E1 -23804.33,E2 -23804.33} C_VEL
LIN {X 0,Y 182.428,Z 1023.53,A -85,B 0,C 180,E1 -23807.611,E2 -23807.611} C_VEL
LIN {X 0,Y 177.099,Z 1030.847,A -85,B 0,C 180,E1 -23810.586,E2 -23810.586} C_VEL
LIN {X 0,Y 172.345,Z 1037.279,A -85,B 0,C 180,E1 -23813.752,E2 -23813.752} C_VEL
LIN {X 0,Y 166.834,Z 1044.545,A -85,B 0,C 180,E1 -23818.227,E2 -23818.227} C_VEL
LIN {X 0,Y 163.356,Z 1049.201,A -85,B 0,C 180,E1 -23821.755,E2 -23821.755} C_VEL
LIN {X 0,Y 159.669,Z 1054.31,A -85,B 0,C 180,E1 -23826.663,E2 -23826.663} C_VEL
LIN {X 0,Y 157.022,Z 1058.323,A -85,B 0,C 180,E1 -23831.742,E2 -23831.742} C_VEL
LIN {X 0,Y 155.366,Z 1061.296,A -85,B 0,C 180,E1 -23836.928,E2 -23836.928} C_VEL
LIN {X 0,Y 154.985,Z 1062.275,A -85,B 0,C 180,E1 -23839.068,E2 -23839.068} C_VEL
LIN {X 0,Y 154.144,Z 1063.133,A -85,B 0,C 180,E1 -23841.209,E2 -23841.209} C_VEL
LIN {X 0,Y 152.528,Z 1063.747,A -85,B 0,C 180,E1 -23843.33,E2 -23843.33} C_VEL
LIN {X 0,Y 148.867,Z 1064.298,A -85,B 0,C 180,E1 -23847.671,E2 -23847.671} C_VEL
LIN {X 0,Y 147.653,Z 1064.223,A -85,B 0,C 180,E1 -23850.725,E2 -23850.725} C_VEL
LIN {X 0,Y 147.521,Z 1063.776,A -85,B 0,C 180,E1 -23855.467,E2 -23855.467} C_VEL
LIN {X 0,Y 147.907,Z 1062.286,A -85,B 0,C 180,E1 -23860.956,E2 -23860.956} C_VEL
LIN {X 0,Y 149.182,Z 1059.798,A -85,B 0,C 180,E1 -23866.419,E2 -23866.419} C_VEL
LIN {X 0,Y 151.653,Z 1056.064,A -85,B 0,C 180,E1 -23872.05,E2 -23872.05} C_VEL
LIN {X 0,Y 154.95,Z 1051.696,A -85,B 0,C 180,E1 -23876.972,E2 -23876.972} C_VEL
LIN {X 0,Y 159.462,Z 1045.96,A -85,B 0,C 180,E1 -23881.929,E2 -23881.929} C_VEL
LIN {X 0,Y 163.638,Z 1040.758,A -85,B 0,C 180,E1 -23885.544,E2 -23885.544} C_VEL
LIN {X 0,Y 169.888,Z 1032.862,A -85,B 0,C 180,E1 -23889.881,E2 -23889.881} C_VEL
LIN {X 0,Y 175.315,Z 1025.882,A -85,B 0,C 180,E1 -23892.959,E2 -23892.959} C_VEL
LIN {X 0,Y 181.141,Z 1017.853,A -85,B 0,C 180,E1 -23895.903,E2 -23895.903} C_VEL
LIN {X 0,Y 187.389,Z 1008.808,A -85,B 0,C 180,E1 -23898.597,E2 -23898.597} C_VEL
LIN {X 0,Y 192.896,Z 1000.244,A -85,B 0,C 180,E1 -23900.733,E2 -23900.733} C_VEL
LIN {X 0,Y 199.981,Z 988.391,A -85,B 0,C 180,E1 -23903.081,E2 -23903.081} C_VEL
LIN {X 0,Y 205.386,Z 978.358,A -85,B 0,C 180,E1 -23904.738,E2 -23904.738} C_VEL
LIN {X 0,Y 211.096,Z 966.572,A -85,B 0,C 180,E1 -23906.336,E2 -23906.336} C_VEL
LIN {X 0,Y 216.295,Z 954.557,A -85,B 0,C 180,E1 -23907.649,E2 -23907.649} C_VEL
LIN {X 0,Y 220.882,Z 942.244,A -85,B 0,C 180,E1 -23908.769,E2 -23908.769} C_VEL
LIN {X 0,Y 224.916,Z 929.708,A -85,B 0,C 180,E1 -23909.676,E2 -23909.676} C_VEL
LIN {X 0,Y 228.519,Z 916.369,A -85,B 0,C 180,E1 -23910.418,E2 -23910.418} C_VEL
LIN {X 0,Y 231.354,Z 903.304,A -85,B 0,C 180,E1 -23910.969,E2 -23910.969} C_VEL
LIN {X 0,Y 233.488,Z 889.514,A -85,B 0,C 180,E1 -23911.434,E2 -23911.434} C_VEL
LIN {X 0,Y 236.372,Z 858.601,A -85,B 0,C 180,E1 -23912.227,E2 -23912.227} C_VEL
LIN {X 0,Y 240.586,Z 810.299,A -85,B 0,C 180,E1 -23913.37,E2 -23913.37} C_VEL
LIN {X 0,Y 236.995,Z 800.73,A -85,B 0,C 180,E1 -23915.82,E2 -23915.82} C_VEL
LIN {X 0,Y 234.163,Z 794.078,A -85,B 0,C 180,E1 -23917.918,E2 -23917.918} C_VEL
LIN {X 0,Y 230.056,Z 786.852,A -85,B 0,C 180,E1 -23921.232,E2 -23921.232} C_VEL
LIN {X 0,Y 227.519,Z 782.74,A -85,B 0,C 180,E1 -23923.628,E2 -23923.628} C_VEL
LIN {X 0,Y 226.024,Z 780.247,A -85,B 0,C 180,E1 -23925.251,E2 -23925.251} C_VEL
LIN {X 0,Y 223.753,Z 776.449,A -85,B 0,C 180,E1 -23928.171,E2 -23928.171} C_VEL
LIN {X 0,Y 221.65,Z 772.931,A -85,B 0,C 180,E1 -23931.796,E2 -23931.796} C_VEL
LIN {X 0,Y 221.257,Z 772.164,A -85,B 0,C 180,E1 -23932.7,E2 -23932.7} C_VEL
LIN {X 0,Y 219.689,Z 769.516,A -85,B 0,C 180,E1 -23940,E2 -23940} C_VEL
LIN {X 0,Y 221.532,Z 772.578,A -85,B 0,C 180,E1 -23948.322,E2 -23948.322} C_VEL
LIN {X 0,Y 223.514,Z 776.207,A -85,B 0,C 180,E1 -23951.908,E2 -23951.908} C_VEL
LIN {X 0,Y 224.391,Z 777.485,A -85,B 0,C 180,E1 -23953.124,E2 -23953.124} C_VEL
LIN {X 0,Y 227.067,Z 781.93,A -85,B 0,C 180,E1 -23956.301,E2 -23956.301} C_VEL
LIN {X 0,Y 229.635,Z 786.172,A -85,B 0,C 180,E1 -23958.802,E2 -23958.802} C_VEL
LIN {X 0,Y 232.754,Z 791.557,A -85,B 0,C 180,E1 -23961.417,E2 -23961.417} C_VEL
LIN {X 0,Y 237.272,Z 799.839,A -85,B 0,C 180,E1 -23964.671,E2 -23964.671} C_VEL
LIN {X 0,Y 246.816,Z 816.47,A -85,B 0,C 180,E1 -23970.123,E2 -23970.123} C_VEL
LIN {X 0,Y 254.425,Z 826.284,A -85,B 0,C 180,E1 -23973.476,E2 -23973.476} C_VEL
LIN {X 0,Y 261.868,Z 834.286,A -85,B 0,C 180,E1 -23976.248,E2 -23976.248} C_VEL
LIN {X 0,Y 277.611,Z 848.204,A -85,B 0,C 180,E1 -23981.043,E2 -23981.043} C_VEL
LIN {X 0,Y 287.455,Z 855.868,A -85,B 0,C 180,E1 -23983.683,E2 -23983.683} C_VEL
LIN {X 0,Y 295.14,Z 861.978,A -85,B 0,C 180,E1 -23985.947,E2 -23985.947} C_VEL
LIN {X 0,Y 301.465,Z 866.824,A -85,B 0,C 180,E1 -23987.948,E2 -23987.948} C_VEL
LIN {X 0,Y 306.546,Z 871.063,A -85,B 0,C 180,E1 -23989.698,E2 -23989.698} C_VEL
LIN {X 0,Y 312.685,Z 875.924,A -85,B 0,C 180,E1 -23991.943,E2 -23991.943} C_VEL
LIN {X 0,Y 318.922,Z 880.922,A -85,B 0,C 180,E1 -23994.378,E2 -23994.378} C_VEL
LIN {X 0,Y 325.888,Z 886.642,A -85,B 0,C 180,E1 -23997.251,E2 -23997.251} C_VEL
LIN {X 0,Y 331.879,Z 891.169,A -85,B 0,C 180,E1 -23999.881,E2 -23999.881} C_VEL
LIN {X 0,Y 336.524,Z 894.953,A -85,B 0,C 180,E1 -24002.056,E2 -24002.056} C_VEL
LIN {X 0,Y 341.701,Z 898.385,A -85,B 0,C 180,E1 -24004.625,E2 -24004.625} C_VEL
LIN {X 0,Y 345.946,Z 901.997,A -85,B 0,C 180,E1 -24006.97,E2 -24006.97} C_VEL
LIN {X 0,Y 350.156,Z 904.995,A -85,B 0,C 180,E1 -24009.495,E2 -24009.495} C_VEL
LIN {X 0,Y 353.867,Z 907.279,A -85,B 0,C 180,E1 -24011.951,E2 -24011.951} C_VEL
LIN {X 0,Y 357.095,Z 910.154,A -85,B 0,C 180,E1 -24014.434,E2 -24014.434} C_VEL
LIN {X 0,Y 360.021,Z 912.292,A -85,B 0,C 180,E1 -24017.039,E2 -24017.039} C_VEL
LIN {X 0,Y 362.25,Z 913.601,A -85,B 0,C 180,E1 -24019.421,E2 -24019.421} C_VEL
LIN {X 0,Y 364.222,Z 914.498,A -85,B 0,C 180,E1 -24021.934,E2 -24021.934} C_VEL
LIN {X 0,Y 365.605,Z 915.1,A -85,B 0,C 180,E1 -24024.485,E2 -24024.485} C_VEL
LIN {X 0,Y 366.455,Z 915.547,A -85,B 0,C 180,E1 -24026.702,E2 -24026.702} C_VEL
LIN {X 0,Y 366.809,Z 915.721,A -85,B 0,C 180,E1 -24028.902,E2 -24028.902} C_VEL
LIN {X 0,Y 366.809,Z 915.721,A -85,B 0,C 180,E1 -24031.098,E2 -24031.098} C_VEL
LIN {X 0,Y 366.258,Z 915.488,A -85,B 0,C 180,E1 -24033.804,E2 -24033.804} C_VEL
LIN {X 0,Y 365.224,Z 914.899,A -85,B 0,C 180,E1 -24036.388,E2 -24036.388} C_VEL
LIN {X 0,Y 363.821,Z 914.22,A -85,B 0,C 180,E1 -24038.606,E2 -24038.606} C_VEL
LIN {X 0,Y 361.746,Z 913.324,A -85,B 0,C 180,E1 -24041.202,E2 -24041.202} C_VEL
LIN {X 0,Y 359.185,Z 911.73,A -85,B 0,C 180,E1 -24043.726,E2 -24043.726} C_VEL
LIN {X 0,Y 355.997,Z 909.271,A -85,B 0,C 180,E1 -24046.428,E2 -24046.428} C_VEL
LIN {X 0,Y 352.948,Z 906.571,A -85,B 0,C 180,E1 -24048.722,E2 -24048.722} C_VEL
LIN {X 0,Y 348.954,Z 904.19,A -85,B 0,C 180,E1 -24051.255,E2 -24051.255} C_VEL
LIN {X 0,Y 344.495,Z 900.816,A -85,B 0,C 180,E1 -24053.843,E2 -24053.843} C_VEL
LIN {X 0,Y 340.6,Z 897.678,A -85,B 0,C 180,E1 -24055.927,E2 -24055.927} C_VEL
LIN {X 0,Y 335.55,Z 894.268,A -85,B 0,C 180,E1 -24058.398,E2 -24058.398} C_VEL
LIN {X 0,Y 329.522,Z 889.278,A -85,B 0,C 180,E1 -24061.175,E2 -24061.175} C_VEL
LIN {X 0,Y 323.989,Z 885.144,A -85,B 0,C 180,E1 -24063.542,E2 -24063.542} C_VEL
LIN {X 0,Y 318.157,Z 880.337,A -85,B 0,C 180,E1 -24065.928,E2 -24065.928} C_VEL
LIN {X 0,Y 311.516,Z 874.875,A -85,B 0,C 180,E1 -24068.509,E2 -24068.509} C_VEL
LIN {X 0,Y 304.203,Z 869.135,A -85,B 0,C 180,E1 -24071.152,E2 -24071.152} C_VEL
LIN {X 0,Y 297.059,Z 863.422,A -85,B 0,C 180,E1 -24073.464,E2 -24073.464} C_VEL
LIN {X 0,Y 290.965,Z 858.467,A -85,B 0,C 180,E1 -24075.305,E2 -24075.305} C_VEL
LIN {X 0,Y 284.419,Z 853.496,A -85,B 0,C 180,E1 -24077.134,E2 -24077.134} C_VEL
LIN {X 0,Y 266.549,Z 838.819,A -85,B 0,C 180,E1 -24082.195,E2 -24082.195} C_VEL
LIN {X 0,Y 255.378,Z 827.435,A -85,B 0,C 180,E1 -24086.142,E2 -24086.142} C_VEL
LIN {X 0,Y 245.964,Z 815.269,A -85,B 0,C 180,E1 -24090.294,E2 -24090.294} C_VEL
LIN {X 0,Y 235.562,Z 796.635,A -85,B 0,C 180,E1 -24096.501,E2 -24096.501} C_VEL
LIN {X 0,Y 231.087,Z 788.631,A -85,B 0,C 180,E1 -24099.935,E2 -24099.935} C_VEL
LIN {X 0,Y 228.016,Z 783.477,A -85,B 0,C 180,E1 -24102.729,E2 -24102.729} C_VEL
LIN {X 0,Y 225.876,Z 780.031,A -85,B 0,C 180,E1 -24105.011,E2 -24105.011} C_VEL
LIN {X 0,Y 223.755,Z 776.451,A -85,B 0,C 180,E1 -24107.76,E2 -24107.76} C_VEL
LIN {X 0,Y 221.721,Z 773.12,A -85,B 0,C 180,E1 -24111.226,E2 -24111.226} C_VEL
LIN {X 0,Y 221.279,Z 772.197,A -85,B 0,C 180,E1 -24112.243,E2 -24112.243} C_VEL
LIN {X 0,Y 219.693,Z 769.485,A -85,B 0,C 180,E1 -24120,E2 -24120} C_VEL
LIN {X 0,Y 221.524,Z 772.544,A -85,B 0,C 180,E1 -24127.893,E2 -24127.893} C_VEL
LIN {X 0,Y 223.423,Z 776.068,A -85,B 0,C 180,E1 -24131.366,E2 -24131.366} C_VEL
LIN {X 0,Y 224.346,Z 777.49,A -85,B 0,C 180,E1 -24132.668,E2 -24132.668} C_VEL
LIN {X 0,Y 227.108,Z 782.026,A -85,B 0,C 180,E1 -24135.941,E2 -24135.941} C_VEL
LIN {X 0,Y 229.591,Z 786.095,A -85,B 0,C 180,E1 -24138.355,E2 -24138.355} C_VEL
LIN {X 0,Y 232.835,Z 791.714,A -85,B 0,C 180,E1 -24141.075,E2 -24141.075} C_VEL
LIN {X 0,Y 234.858,Z 795.542,A -85,B 0,C 180,E1 -24142.606,E2 -24142.606} C_VEL
LIN {X 0,Y 238.623,Z 804.935,A -85,B 0,C 180,E1 -24145.318,E2 -24145.318} C_VEL
LIN {X 0,Y 240.589,Z 810.275,A -85,B 0,C 180,E1 -24146.629,E2 -24146.629} C_VEL
LIN {X 0,Y 233.726,Z 887.418,A -85,B 0,C 180,E1 -24148.488,E2 -24148.488} C_VEL
LIN {X 0,Y 231.874,Z 900.24,A -85,B 0,C 180,E1 -24148.912,E2 -24148.912} C_VEL
LIN {X 0,Y 229.39,Z 912.591,A -85,B 0,C 180,E1 -24149.402,E2 -24149.402} C_VEL
LIN {X 0,Y 226.319,Z 924.927,A -85,B 0,C 180,E1 -24150.049,E2 -24150.049} C_VEL
LIN {X 0,Y 222.864,Z 936.303,A -85,B 0,C 180,E1 -24150.762,E2 -24150.762} C_VEL
LIN {X 0,Y 218.266,Z 949.534,A -85,B 0,C 180,E1 -24151.872,E2 -24151.872} C_VEL
LIN {X 0,Y 213.016,Z 962.261,A -85,B 0,C 180,E1 -24153.158,E2 -24153.158} C_VEL
LIN {X 0,Y 207.92,Z 973.249,A -85,B 0,C 180,E1 -24154.524,E2 -24154.524} C_VEL
LIN {X 0,Y 202.362,Z 984.045,A -85,B 0,C 180,E1 -24156.154,E2 -24156.154} C_VEL
LIN {X 0,Y 196.456,Z 994.534,A -85,B 0,C 180,E1 -24158.094,E2 -24158.094} C_VEL
LIN {X 0,Y 190.687,Z 1003.795,A -85,B 0,C 180,E1 -24160.116,E2 -24160.116} C_VEL
LIN {X 0,Y 184.165,Z 1013.521,A -85,B 0,C 180,E1 -24162.728,E2 -24162.728} C_VEL
LIN {X 0,Y 178.114,Z 1022.041,A -85,B 0,C 180,E1 -24165.544,E2 -24165.544} C_VEL
LIN {X 0,Y 171.602,Z 1030.639,A -85,B 0,C 180,E1 -24169.06,E2 -24169.06} C_VEL
LIN {X 0,Y 166.577,Z 1037.07,A -85,B 0,C 180,E1 -24172.284,E2 -24172.284} C_VEL
LIN {X 0,Y 162.111,Z 1042.713,A -85,B 0,C 180,E1 -24175.697,E2 -24175.697} C_VEL
LIN {X 0,Y 157.034,Z 1048.992,A -85,B 0,C 180,E1 -24180.509,E2 -24180.509} C_VEL
LIN {X 0,Y 153.085,Z 1054.102,A -85,B 0,C 180,E1 -24185.596,E2 -24185.596} C_VEL
LIN {X 0,Y 150.206,Z 1058.115,A -85,B 0,C 180,E1 -24190.882,E2 -24190.882} C_VEL
LIN {X 0,Y 148.383,Z 1061.089,A -85,B 0,C 180,E1 -24196.301,E2 -24196.301} C_VEL
LIN {X 0,Y 147.907,Z 1062.286,A -85,B 0,C 180,E1 -24199.044,E2 -24199.044} C_VEL
LIN {X 0,Y 147.521,Z 1063.776,A -85,B 0,C 180,E1 -24204.533,E2 -24204.533} C_VEL
LIN {X 0,Y 147.717,Z 1064.279,A -85,B 0,C 180,E1 -24210,E2 -24210} C_VEL
LIN {X 0,Y 147.653,Z 1064.223,A -85,B 0,C 180,E1 -24210.725,E2 -24210.725} C_VEL
LIN {X 0,Y 146.86,Z 1064.022,A -85,B 0,C 180,E1 -24213,E2 -24213} C_VEL
LIN {X 0,Y 145.235,Z 1063.763,A -85,B 0,C 180,E1 -24215.242,E2 -24215.242} C_VEL
LIN {X 0,Y 141.756,Z 1062.598,A -85,B 0,C 180,E1 -24219.809,E2 -24219.809} C_VEL
LIN {X 0,Y 141.041,Z 1061.807,A -85,B 0,C 180,E1 -24222.19,E2 -24222.19} C_VEL
LIN {X 0,Y 141.104,Z 1061.465,A -85,B 0,C 180,E1 -24222.988,E2 -24222.988} C_VEL
LIN {X 0,Y 142.305,Z 1059.59,A -85,B 0,C 180,E1 -24227.236,E2 -24227.236} C_VEL
LIN {X 0,Y 145.68,Z 1054.985,A -85,B 0,C 180,E1 -24234.208,E2 -24234.208} C_VEL
LIN {X 0,Y 148.545,Z 1051.486,A -85,B 0,C 180,E1 -24238.236,E2 -24238.236} C_VEL
LIN {X 0,Y 153.37,Z 1045.751,A -85,B 0,C 180,E1 -24243.358,E2 -24243.358} C_VEL
LIN {X 0,Y 158.429,Z 1039.826,A -85,B 0,C 180,E1 -24247.505,E2 -24247.505} C_VEL
LIN {X 0,Y 164.421,Z 1032.654,A -85,B 0,C 180,E1 -24251.492,E2 -24251.492} C_VEL
LIN {X 0,Y 170.109,Z 1025.674,A -85,B 0,C 180,E1 -24254.614,E2 -24254.614} C_VEL
LIN {X 0,Y 175.956,Z 1018,A -85,B 0,C 180,E1 -24257.469,E2 -24257.469} C_VEL
LIN {X 0,Y 182.707,Z 1008.599,A -85,B 0,C 180,E1 -24260.291,E2 -24260.291} C_VEL
LIN {X 0,Y 188.442,Z 1000.036,A -85,B 0,C 180,E1 -24262.42,E2 -24262.42} C_VEL
LIN {X 0,Y 195.379,Z 988.862,A -85,B 0,C 180,E1 -24264.638,E2 -24264.638} C_VEL
LIN {X 0,Y 201.339,Z 978.151,A -85,B 0,C 180,E1 -24266.401,E2 -24266.401} C_VEL
LIN {X 0,Y 207.23,Z 966.366,A -85,B 0,C 180,E1 -24267.976,E2 -24267.976} C_VEL
LIN {X 0,Y 212.572,Z 954.351,A -85,B 0,C 180,E1 -24269.27,E2 -24269.27} C_VEL
LIN {X 0,Y 217.269,Z 942.038,A -85,B 0,C 180,E1 -24270.378,E2 -24270.378} C_VEL
LIN {X 0,Y 221.417,Z 929.503,A -85,B 0,C 180,E1 -24271.261,E2 -24271.261} C_VEL
LIN {X 0,Y 225.091,Z 916.218,A -85,B 0,C 180,E1 -24271.985,E2 -24271.985} C_VEL
LIN {X 0,Y 227.893,Z 903.648,A -85,B 0,C 180,E1 -24272.51,E2 -24272.51} C_VEL
LIN {X 0,Y 230.105,Z 889.898,A -85,B 0,C 180,E1 -24272.972,E2 -24272.972} C_VEL
LIN {X 0,Y 232.824,Z 861.936,A -85,B 0,C 180,E1 -24273.692,E2 -24273.692} C_VEL
LIN {X 0,Y 237.161,Z 813.312,A -85,B 0,C 180,E1 -24274.845,E2 -24274.845} C_VEL
LIN {X 0,Y 233.431,Z 803.242,A -85,B 0,C 180,E1 -24277.63,E2 -24277.63} C_VEL
LIN {X 0,Y 231.894,Z 799.782,A -85,B 0,C 180,E1 -24278.848,E2 -24278.848} C_VEL
LIN {X 0,Y 228.508,Z 793.483,A -85,B 0,C 180,E1 -24281.74,E2 -24281.74} C_VEL
LIN {X 0,Y 226.109,Z 789.46,A -85,B 0,C 180,E1 -24284.102,E2 -24284.102} C_VEL
LIN {X 0,Y 224.411,Z 786.559,A -85,B 0,C 180,E1 -24286.046,E2 -24286.046} C_VEL
LIN {X 0,Y 222.554,Z 783.266,A -85,B 0,C 180,E1 -24288.592,E2 -24288.592} C_VEL
LIN {X 0,Y 220.525,Z 779.631,A -85,B 0,C 180,E1 -24292.33,E2 -24292.33} C_VEL
LIN {X 0,Y 220.192,Z 779.075,A -85,B 0,C 180,E1 -24293.125,E2 -24293.125} C_VEL
LIN {X 0,Y 218.82,Z 776.596,A -85,B 0,C 180,E1 -24300,E2 -24300} C_VEL
LIN {X 0,Y 220.458,Z 779.422,A -85,B 0,C 180,E1 -24307.901,E2 -24307.901} C_VEL
LIN {X 0,Y 222.237,Z 782.917,A -85,B 0,C 180,E1 -24311.353,E2 -24311.353} C_VEL
LIN {X 0,Y 223.115,Z 784.22,A -85,B 0,C 180,E1 -24312.636,E2 -24312.636} C_VEL
LIN {X 0,Y 225.826,Z 788.912,A -85,B 0,C 180,E1 -24315.992,E2 -24315.992} C_VEL
LIN {X 0,Y 228.177,Z 792.943,A -85,B 0,C 180,E1 -24318.364,E2 -24318.364} C_VEL
LIN {X 0,Y 231.827,Z 799.672,A -85,B 0,C 180,E1 -24321.507,E2 -24321.507} C_VEL
LIN {X 0,Y 235.177,Z 806.088,A -85,B 0,C 180,E1 -24323.992,E2 -24323.992} C_VEL
LIN {X 0,Y 244.334,Z 822.465,A -85,B 0,C 180,E1 -24329.451,E2 -24329.451} C_VEL
LIN {X 0,Y 251.777,Z 832.28,A -85,B 0,C 180,E1 -24332.858,E2 -24332.858} C_VEL
LIN {X 0,Y 259.065,Z 840.286,A -85,B 0,C 180,E1 -24335.669,E2 -24335.669} C_VEL
LIN {X 0,Y 268.805,Z 849.24,A -85,B 0,C 180,E1 -24338.864,E2 -24338.864} C_VEL
LIN {X 0,Y 284.107,Z 861.627,A -85,B 0,C 180,E1 -24343.106,E2 -24343.106} C_VEL
LIN {X 0,Y 292.761,Z 868.329,A -85,B 0,C 180,E1 -24345.551,E2 -24345.551} C_VEL
LIN {X 0,Y 300.139,Z 874.05,A -85,B 0,C 180,E1 -24347.859,E2 -24347.859} C_VEL
LIN {X 0,Y 306.707,Z 879.288,A -85,B 0,C 180,E1 -24350.113,E2 -24350.113} C_VEL
LIN {X 0,Y 313.099,Z 884.457,A -85,B 0,C 180,E1 -24352.496,E2 -24352.496} C_VEL
LIN {X 0,Y 320.101,Z 889.971,A -85,B 0,C 180,E1 -24355.252,E2 -24355.252} C_VEL
LIN {X 0,Y 326.347,Z 894.98,A -85,B 0,C 180,E1 -24357.874,E2 -24357.874} C_VEL
LIN {X 0,Y 330.648,Z 898.196,A -85,B 0,C 180,E1 -24359.755,E2 -24359.755} C_VEL
LIN {X 0,Y 335.414,Z 901.994,A -85,B 0,C 180,E1 -24361.975,E2 -24361.975} C_VEL
LIN {X 0,Y 340.351,Z 905.255,A -85,B 0,C 180,E1 -24364.41,E2 -24364.41} C_VEL
LIN {X 0,Y 344.695,Z 908.902,A -85,B 0,C 180,E1 -24366.793,E2 -24366.793} C_VEL
LIN {X 0,Y 348.906,Z 911.863,A -85,B 0,C 180,E1 -24369.285,E2 -24369.285} C_VEL
LIN {X 0,Y 352.806,Z 914.285,A -85,B 0,C 180,E1 -24371.835,E2 -24371.835} C_VEL
LIN {X 0,Y 356.112,Z 917.17,A -85,B 0,C 180,E1 -24374.35,E2 -24374.35} C_VEL
LIN {X 0,Y 358.917,Z 919.214,A -85,B 0,C 180,E1 -24376.843,E2 -24376.843} C_VEL
LIN {X 0,Y 361.352,Z 920.645,A -85,B 0,C 180,E1 -24379.394,E2 -24379.394} C_VEL
LIN {X 0,Y 363.339,Z 921.543,A -85,B 0,C 180,E1 -24381.914,E2 -24381.914} C_VEL
LIN {X 0,Y 364.73,Z 922.143,A -85,B 0,C 180,E1 -24384.471,E2 -24384.471} C_VEL
LIN {X 0,Y 365.586,Z 922.593,A -85,B 0,C 180,E1 -24386.694,E2 -24386.694} C_VEL
LIN {X 0,Y 365.942,Z 922.767,A -85,B 0,C 180,E1 -24388.9,E2 -24388.9} C_VEL
LIN {X 0,Y 365.942,Z 922.768,A -85,B 0,C 180,E1 -24391.1,E2 -24391.1} C_VEL
LIN {X 0,Y 365.586,Z 922.594,A -85,B 0,C 180,E1 -24393.306,E2 -24393.306} C_VEL
LIN {X 0,Y 364.725,Z 922.187,A -85,B 0,C 180,E1 -24395.529,E2 -24395.529} C_VEL
LIN {X 0,Y 364.216,Z 921.793,A -85,B 0,C 180,E1 -24396.648,E2 -24396.648} C_VEL
LIN {X 0,Y 362.931,Z 921.263,A -85,B 0,C 180,E1 -24398.627,E2 -24398.627} C_VEL
LIN {X 0,Y 360.844,Z 920.363,A -85,B 0,C 180,E1 -24401.231,E2 -24401.231} C_VEL
LIN {X 0,Y 358.262,Z 918.786,A -85,B 0,C 180,E1 -24403.762,E2 -24403.762} C_VEL
LIN {X 0,Y 355.045,Z 916.316,A -85,B 0,C 180,E1 -24406.474,E2 -24406.474} C_VEL
LIN {X 0,Y 351.747,Z 913.468,A -85,B 0,C 180,E1 -24408.911,E2 -24408.911} C_VEL
LIN {X 0,Y 347.731,Z 911.063,A -85,B 0,C 180,E1 -24411.456,E2 -24411.456} C_VEL
LIN {X 0,Y 343.202,Z 907.677,A -85,B 0,C 180,E1 -24414.057,E2 -24414.057} C_VEL
LIN {X 0,Y 339.486,Z 904.674,A -85,B 0,C 180,E1 -24416.019,E2 -24416.019} C_VEL
LIN {X 0,Y 334.131,Z 901.106,A -85,B 0,C 180,E1 -24418.617,E2 -24418.617} C_VEL
LIN {X 0,Y 327.903,Z 895.985,A -85,B 0,C 180,E1 -24421.471,E2 -24421.471} C_VEL
LIN {X 0,Y 322.375,Z 891.89,A -85,B 0,C 180,E1 -24423.81,E2 -24423.81} C_VEL
LIN {X 0,Y 316.476,Z 887.078,A -85,B 0,C 180,E1 -24426.192,E2 -24426.192} C_VEL
LIN {X 0,Y 309.801,Z 881.64,A -85,B 0,C 180,E1 -24428.762,E2 -24428.762} C_VEL
LIN {X 0,Y 302.608,Z 876.1,A -85,B 0,C 180,E1 -24431.32,E2 -24431.32} C_VEL
LIN {X 0,Y 296.73,Z 871.358,A -85,B 0,C 180,E1 -24433.224,E2 -24433.224} C_VEL
LIN {X 0,Y 290.26,Z 866.338,A -85,B 0,C 180,E1 -24435.167,E2 -24435.167} C_VEL
LIN {X 0,Y 283.171,Z 860.917,A -85,B 0,C 180,E1 -24437.142,E2 -24437.142} C_VEL
LIN {X 0,Y 263.278,Z 844.44,A -85,B 0,C 180,E1 -24442.878,E2 -24442.878} C_VEL
LIN {X 0,Y 252.679,Z 833.358,A -85,B 0,C 180,E1 -24446.769,E2 -24446.769} C_VEL
LIN {X 0,Y 245.464,Z 824.05,A -85,B 0,C 180,E1 -24449.99,E2 -24449.99} C_VEL
LIN {X 0,Y 238.472,Z 812.67,A -85,B 0,C 180,E1 -24453.825,E2 -24453.825} C_VEL
LIN {X 0,Y 233.452,Z 802.684,A -85,B 0,C 180,E1 -24457.254,E2 -24457.254} C_VEL
LIN {X 0,Y 229.191,Z 794.745,A -85,B 0,C 180,E1 -24460.709,E2 -24460.709} C_VEL
LIN {X 0,Y 226.471,Z 790.021,A -85,B 0,C 180,E1 -24463.319,E2 -24463.319} C_VEL
LIN {X 0,Y 224.436,Z 786.6,A -85,B 0,C 180,E1 -24465.609,E2 -24465.609} C_VEL
LIN {X 0,Y 222.653,Z 783.375,A -85,B 0,C 180,E1 -24468.046,E2 -24468.046} C_VEL
LIN {X 0,Y 220.709,Z 780.128,A -85,B 0,C 180,E1 -24471.474,E2 -24471.474} C_VEL
LIN {X 0,Y 220.417,Z 779.285,A -85,B 0,C 180,E1 -24472.212,E2 -24472.212} C_VEL
LIN {X 0,Y 218.823,Z 776.57,A -85,B 0,C 180,E1 -24480,E2 -24480} C_VEL
LIN {X 0,Y 220.483,Z 779.487,A -85,B 0,C 180,E1 -24487.556,E2 -24487.556} C_VEL
LIN {X 0,Y 222.396,Z 783.055,A -85,B 0,C 180,E1 -24491.174,E2 -24491.174} C_VEL
LIN {X 0,Y 223.523,Z 785.103,A -85,B 0,C 180,E1 -24492.819,E2 -24492.819} C_VEL
LIN {X 0,Y 225.615,Z 788.568,A -85,B 0,C 180,E1 -24495.354,E2 -24495.354} C_VEL
LIN {X 0,Y 228.274,Z 793.116,A -85,B 0,C 180,E1 -24498.048,E2 -24498.048} C_VEL
LIN {X 0,Y 231.764,Z 799.522,A -85,B 0,C 180,E1 -24501.048,E2 -24501.048} C_VEL
LIN {X 0,Y 233.29,Z 802.919,A -85,B 0,C 180,E1 -24502.261,E2 -24502.261} C_VEL
LIN {X 0,Y 236.996,Z 812.905,A -85,B 0,C 180,E1 -24505.042,E2 -24505.042} C_VEL
LIN {X 0,Y 237.205,Z 813.529,A -85,B 0,C 180,E1 -24505.192,E2 -24505.192} C_VEL
LIN {X 0,Y 230.339,Z 887.94,A -85,B 0,C 180,E1 -24506.96,E2 -24506.96} C_VEL
LIN {X 0,Y 228.251,Z 901.54,A -85,B 0,C 180,E1 -24507.405,E2 -24507.405} C_VEL
LIN {X 0,Y 225.623,Z 913.974,A -85,B 0,C 180,E1 -24507.911,E2 -24507.911} C_VEL
LIN {X 0,Y 222.49,Z 925.917,A -85,B 0,C 180,E1 -24508.536,E2 -24508.536} C_VEL
LIN {X 0,Y 219.317,Z 936.098,A -85,B 0,C 180,E1 -24509.167,E2 -24509.167} C_VEL
LIN {X 0,Y 214.593,Z 949.328,A -85,B 0,C 180,E1 -24510.258,E2 -24510.258} C_VEL
LIN {X 0,Y 209.212,Z 962.055,A -85,B 0,C 180,E1 -24511.527,E2 -24511.527} C_VEL
LIN {X 0,Y 203.967,Z 973.043,A -85,B 0,C 180,E1 -24512.875,E2 -24512.875} C_VEL
LIN {X 0,Y 198.236,Z 983.839,A -85,B 0,C 180,E1 -24514.489,E2 -24514.489} C_VEL
LIN {X 0,Y 192.113,Z 994.327,A -85,B 0,C 180,E1 -24516.409,E2 -24516.409} C_VEL
LIN {X 0,Y 186.144,Z 1003.587,A -85,B 0,C 180,E1 -24518.426,E2 -24518.426} C_VEL
LIN {X 0,Y 179.364,Z 1013.312,A -85,B 0,C 180,E1 -24521.04,E2 -24521.04} C_VEL
LIN {X 0,Y 173.061,Z 1021.834,A -85,B 0,C 180,E1 -24523.879,E2 -24523.879} C_VEL
LIN {X 0,Y 166.238,Z 1030.431,A -85,B 0,C 180,E1 -24527.436,E2 -24527.436} C_VEL
LIN {X 0,Y 160.948,Z 1036.862,A -85,B 0,C 180,E1 -24530.717,E2 -24530.717} C_VEL
LIN {X 0,Y 156.19,Z 1042.503,A -85,B 0,C 180,E1 -24534.201,E2 -24534.201} C_VEL
LIN {X 0,Y 150.803,Z 1048.784,A -85,B 0,C 180,E1 -24539.161,E2 -24539.161} C_VEL
LIN {X 0,Y 146.548,Z 1053.893,A -85,B 0,C 180,E1 -24544.431,E2 -24544.431} C_VEL
LIN {X 0,Y 143.432,Z 1057.907,A -85,B 0,C 180,E1 -24549.941,E2 -24549.941} C_VEL
LIN {X 0,Y 141.417,Z 1060.881,A -85,B 0,C 180,E1 -24555.613,E2 -24555.613} C_VEL
LIN {X 0,Y 140.867,Z 1062.079,A -85,B 0,C 180,E1 -24558.489,E2 -24558.489} C_VEL
LIN {X 0,Y 140.427,Z 1063.57,A -85,B 0,C 180,E1 -24564.256,E2 -24564.256} C_VEL
LIN {X 0,Y 140.629,Z 1064.074,A -85,B 0,C 180,E1 -24570,E2 -24570} C_VEL
LIN {X 0,Y 140.427,Z 1063.57,A -85,B 0,C 180,E1 -24575.744,E2 -24575.744} C_VEL
LIN {X 0,Y 140.866,Z 1062.079,A -85,B 0,C 180,E1 -24581.511,E2 -24581.511} C_VEL
LIN {X 0,Y 141.104,Z 1061.465,A -85,B 0,C 180,E1 -24582.988,E2 -24582.988} C_VEL
LIN {X 0,Y 140.995,Z 1060.511,A -85,B 0,C 180,E1 -24585.352,E2 -24585.352} C_VEL
LIN {X 0,Y 139.472,Z 1058.557,A -85,B 0,C 180,E1 -24589.283,E2 -24589.283} C_VEL
LIN {X 0,Y 138.524,Z 1056.838,A -85,B 0,C 180,E1 -24592.461,E2 -24592.461} C_VEL
LIN {X 0,Y 138.827,Z 1055.235,A -85,B 0,C 180,E1 -24594.822,E2 -24594.822} C_VEL
LIN {X 0,Y 139.231,Z 1054.655,A -85,B 0,C 180,E1 -24595.586,E2 -24595.586} C_VEL
LIN {X 0,Y 142.232,Z 1051.278,A -85,B 0,C 180,E1 -24599.611,E2 -24599.611} C_VEL
LIN {X 0,Y 147.386,Z 1045.541,A -85,B 0,C 180,E1 -24604.903,E2 -24604.903} C_VEL
LIN {X 0,Y 152.029,Z 1040.478,A -85,B 0,C 180,E1 -24608.613,E2 -24608.613} C_VEL
LIN {X 0,Y 159.094,Z 1032.445,A -85,B 0,C 180,E1 -24613.212,E2 -24613.212} C_VEL
LIN {X 0,Y 165.061,Z 1025.465,A -85,B 0,C 180,E1 -24616.37,E2 -24616.37} C_VEL
LIN {X 0,Y 171.405,Z 1017.499,A -85,B 0,C 180,E1 -24619.334,E2 -24619.334} C_VEL
LIN {X 0,Y 178.206,Z 1008.392,A -85,B 0,C 180,E1 -24622.067,E2 -24622.067} C_VEL
LIN {X 0,Y 184.162,Z 999.829,A -85,B 0,C 180,E1 -24624.186,E2 -24624.186} C_VEL
LIN {X 0,Y 191.824,Z 987.751,A -85,B 0,C 180,E1 -24626.557,E2 -24626.557} C_VEL
LIN {X 0,Y 198.196,Z 976.573,A -85,B 0,C 180,E1 -24628.322,E2 -24628.322} C_VEL
LIN {X 0,Y 203.539,Z 966.16,A -85,B 0,C 180,E1 -24629.678,E2 -24629.678} C_VEL
LIN {X 0,Y 209.021,Z 954.145,A -85,B 0,C 180,E1 -24630.948,E2 -24630.948} C_VEL
LIN {X 0,Y 213.831,Z 941.832,A -85,B 0,C 180,E1 -24632.04,E2 -24632.04} C_VEL
LIN {X 0,Y 218.087,Z 929.297,A -85,B 0,C 180,E1 -24632.9,E2 -24632.9} C_VEL
LIN {X 0,Y 221.885,Z 915.8,A -85,B 0,C 180,E1 -24633.619,E2 -24633.619} C_VEL
LIN {X 0,Y 224.725,Z 903.327,A -85,B 0,C 180,E1 -24634.121,E2 -24634.121} C_VEL
LIN {X 0,Y 227.012,Z 889.32,A -85,B 0,C 180,E1 -24634.579,E2 -24634.579} C_VEL
LIN {X 0,Y 229.849,Z 860.833,A -85,B 0,C 180,E1 -24635.299,E2 -24635.299} C_VEL
LIN {X 0,Y 233.888,Z 816.526,A -85,B 0,C 180,E1 -24636.353,E2 -24636.353} C_VEL
LIN {X 0,Y 230.681,Z 807.584,A -85,B 0,C 180,E1 -24638.965,E2 -24638.965} C_VEL
LIN {X 0,Y 228.407,Z 802.898,A -85,B 0,C 180,E1 -24640.917,E2 -24640.917} C_VEL
LIN {X 0,Y 225.649,Z 797.657,A -85,B 0,C 180,E1 -24643.593,E2 -24643.593} C_VEL
LIN {X 0,Y 222.999,Z 793.11,A -85,B 0,C 180,E1 -24646.653,E2 -24646.653} C_VEL
LIN {X 0,Y 221.368,Z 790.082,A -85,B 0,C 180,E1 -24649.018,E2 -24649.018} C_VEL
LIN {X 0,Y 219.5,Z 786.592,A -85,B 0,C 180,E1 -24652.641,E2 -24652.641} C_VEL
LIN {X 0,Y 218.967,Z 785.787,A -85,B 0,C 180,E1 -24654.012,E2 -24654.012} C_VEL
LIN {X 0,Y 217.95,Z 783.679,A -85,B 0,C 180,E1 -24660,E2 -24660} C_VEL
LIN {X 0,Y 219.437,Z 786.392,A -85,B 0,C 180,E1 -24667.591,E2 -24667.591} C_VEL
LIN {X 0,Y 221.401,Z 790.142,A -85,B 0,C 180,E1 -24671.443,E2 -24671.443} C_VEL
LIN {X 0,Y 224.189,Z 795.144,A -85,B 0,C 180,E1 -24675.212,E2 -24675.212} C_VEL
LIN {X 0,Y 227.226,Z 800.568,A -85,B 0,C 180,E1 -24678.39,E2 -24678.39} C_VEL
LIN {X 0,Y 231.904,Z 809.709,A -85,B 0,C 180,E1 -24682.377,E2 -24682.377} C_VEL
LIN {X 0,Y 241.921,Z 828.51,A -85,B 0,C 180,E1 -24688.783,E2 -24688.783} C_VEL
LIN {X 0,Y 249.283,Z 838.429,A -85,B 0,C 180,E1 -24692.281,E2 -24692.281} C_VEL
LIN {X 0,Y 256.444,Z 846.446,A -85,B 0,C 180,E1 -24695.135,E2 -24695.135} C_VEL
LIN {X 0,Y 272.702,Z 861.108,A -85,B 0,C 180,E1 -24700.354,E2 -24700.354} C_VEL
LIN {X 0,Y 284.759,Z 870.347,A -85,B 0,C 180,E1 -24703.591,E2 -24703.591} C_VEL
LIN {X 0,Y 293.089,Z 876.816,A -85,B 0,C 180,E1 -24706.002,E2 -24706.002} C_VEL
LIN {X 0,Y 299.756,Z 882.087,A -85,B 0,C 180,E1 -24708.14,E2 -24708.14} C_VEL
LIN {X 0,Y 306.539,Z 887.244,A -85,B 0,C 180,E1 -24710.491,E2 -24710.491} C_VEL
LIN {X 0,Y 313.54,Z 892.926,A -85,B 0,C 180,E1 -24713.108,E2 -24713.108} C_VEL
LIN {X 0,Y 318.981,Z 897.25,A -85,B 0,C 180,E1 -24715.255,E2 -24715.255} C_VEL
LIN {X 0,Y 325.175,Z 902.074,A -85,B 0,C 180,E1 -24717.821,E2 -24717.821} C_VEL
LIN {X 0,Y 329.026,Z 904.992,A -85,B 0,C 180,E1 -24719.517,E2 -24719.517} C_VEL
LIN {X 0,Y 333.695,Z 908.684,A -85,B 0,C 180,E1 -24721.684,E2 -24721.684} C_VEL
LIN {X 0,Y 338.848,Z 912.087,A -85,B 0,C 180,E1 -24724.18,E2 -24724.18} C_VEL
LIN {X 0,Y 343.335,Z 915.794,A -85,B 0,C 180,E1 -24726.623,E2 -24726.623} C_VEL
LIN {X 0,Y 347.758,Z 918.874,A -85,B 0,C 180,E1 -24729.214,E2 -24729.214} C_VEL
LIN {X 0,Y 351.43,Z 921.092,A -85,B 0,C 180,E1 -24731.602,E2 -24731.602} C_VEL
LIN {X 0,Y 354.721,Z 923.989,A -85,B 0,C 180,E1 -24734.092,E2 -24734.092} C_VEL
LIN {X 0,Y 357.828,Z 926.232,A -85,B 0,C 180,E1 -24736.803,E2 -24736.803} C_VEL
LIN {X 0,Y 360.253,Z 927.656,A -85,B 0,C 180,E1 -24739.362,E2 -24739.362} C_VEL
LIN {X 0,Y 362.167,Z 928.479,A -85,B 0,C 180,E1 -24741.755,E2 -24741.755} C_VEL
LIN {X 0,Y 363.702,Z 929.16,A -85,B 0,C 180,E1 -24744.456,E2 -24744.456} C_VEL
LIN {X 0,Y 364.537,Z 929.605,A -85,B 0,C 180,E1 -24746.684,E2 -24746.684} C_VEL
LIN {X 0,Y 364.927,Z 929.794,A -85,B 0,C 180,E1 -24748.897,E2 -24748.897} C_VEL
LIN {X 0,Y 364.926,Z 929.794,A -85,B 0,C 180,E1 -24751.103,E2 -24751.103} C_VEL
LIN {X 0,Y 364.537,Z 929.603,A -85,B 0,C 180,E1 -24753.316,E2 -24753.316} C_VEL
LIN {X 0,Y 363.694,Z 929.211,A -85,B 0,C 180,E1 -24755.544,E2 -24755.544} C_VEL
LIN {X 0,Y 362.462,Z 928.652,A -85,B 0,C 180,E1 -24757.8,E2 -24757.8} C_VEL
LIN {X 0,Y 360.751,Z 927.874,A -85,B 0,C 180,E1 -24760.098,E2 -24760.098} C_VEL
LIN {X 0,Y 358.412,Z 926.619,A -85,B 0,C 180,E1 -24762.634,E2 -24762.634} C_VEL
LIN {X 0,Y 355.487,Z 924.581,A -85,B 0,C 180,E1 -24765.26,E2 -24765.26} C_VEL
LIN {X 0,Y 352.344,Z 921.933,A -85,B 0,C 180,E1 -24767.744,E2 -24767.744} C_VEL
LIN {X 0,Y 350.407,Z 920.353,A -85,B 0,C 180,E1 -24769.11,E2 -24769.11} C_VEL
LIN {X 0,Y 346.157,Z 917.799,A -85,B 0,C 180,E1 -24771.767,E2 -24771.767} C_VEL
LIN {X 0,Y 341.678,Z 914.456,A -85,B 0,C 180,E1 -24774.291,E2 -24774.291} C_VEL
LIN {X 0,Y 337.854,Z 911.443,A -85,B 0,C 180,E1 -24776.32,E2 -24776.32} C_VEL
LIN {X 0,Y 332.177,Z 907.585,A -85,B 0,C 180,E1 -24779.029,E2 -24779.029} C_VEL
LIN {X 0,Y 326.271,Z 902.755,A -85,B 0,C 180,E1 -24781.721,E2 -24781.721} C_VEL
LIN {X 0,Y 320.487,Z 898.501,A -85,B 0,C 180,E1 -24784.108,E2 -24784.108} C_VEL
LIN {X 0,Y 314.164,Z 893.384,A -85,B 0,C 180,E1 -24786.654,E2 -24786.654} C_VEL
LIN {X 0,Y 307.249,Z 887.805,A -85,B 0,C 180,E1 -24789.253,E2 -24789.253} C_VEL
LIN {X 0,Y 300.241,Z 882.501,A -85,B 0,C 180,E1 -24791.695,E2 -24791.695} C_VEL
LIN {X 0,Y 293.342,Z 877.003,A -85,B 0,C 180,E1 -24793.92,E2 -24793.92} C_VEL
LIN {X 0,Y 285.551,Z 870.896,A -85,B 0,C 180,E1 -24796.195,E2 -24796.195} C_VEL
LIN {X 0,Y 275.892,Z 863.484,A -85,B 0,C 180,E1 -24798.775,E2 -24798.775} C_VEL
LIN {X 0,Y 260.047,Z 850.042,A -85,B 0,C 180,E1 -24803.579,E2 -24803.579} C_VEL
LIN {X 0,Y 249.989,Z 839.301,A -85,B 0,C 180,E1 -24807.416,E2 -24807.416} C_VEL
LIN {X 0,Y 242.715,Z 829.648,A -85,B 0,C 180,E1 -24810.807,E2 -24810.807} C_VEL
LIN {X 0,Y 235.578,Z 817.463,A -85,B 0,C 180,E1 -24814.967,E2 -24814.967} C_VEL
LIN {X 0,Y 231.497,Z 808.942,A -85,B 0,C 180,E1 -24817.934,E2 -24817.934} C_VEL
LIN {X 0,Y 227.531,Z 801.221,A -85,B 0,C 180,E1 -24821.314,E2 -24821.314} C_VEL
LIN {X 0,Y 225.066,Z 796.735,A -85,B 0,C 180,E1 -24823.795,E2 -24823.795} C_VEL
LIN {X 0,Y 223.025,Z 793.137,A -85,B 0,C 180,E1 -24826.214,E2 -24826.214} C_VEL
LIN {X 0,Y 221.258,Z 789.925,A -85,B 0,C 180,E1 -24828.782,E2 -24828.782} C_VEL
LIN {X 0,Y 219.479,Z 786.517,A -85,B 0,C 180,E1 -24832.295,E2 -24832.295} C_VEL
LIN {X 0,Y 218.296,Z 785.074,A -85,B 0,C 180,E1 -24835.846,E2 -24835.846} C_VEL
LIN {X 0,Y 217.954,Z 783.648,A -85,B 0,C 180,E1 -24840,E2 -24840} C_VEL
LIN {X 0,Y 219.461,Z 786.442,A -85,B 0,C 180,E1 -24847.244,E2 -24847.244} C_VEL
LIN {X 0,Y 221.873,Z 791.056,A -85,B 0,C 180,E1 -24851.773,E2 -24851.773} C_VEL
LIN {X 0,Y 224.43,Z 795.613,A -85,B 0,C 180,E1 -24855.089,E2 -24855.089} C_VEL
LIN {X 0,Y 227.312,Z 800.766,A -85,B 0,C 180,E1 -24858.068,E2 -24858.068} C_VEL
LIN {X 0,Y 230.437,Z 806.956,A -85,B 0,C 180,E1 -24860.824,E2 -24860.824} C_VEL
LIN {X 0,Y 233.639,Z 815.792,A -85,B 0,C 180,E1 -24863.453,E2 -24863.453} C_VEL
LIN {X 0,Y 233.946,Z 816.658,A -85,B 0,C 180,E1 -24863.688,E2 -24863.688} C_VEL
LIN {X 0,Y 227.225,Z 887.562,A -85,B 0,C 180,E1 -24865.355,E2 -24865.355} C_VEL
LIN {X 0,Y 225.072,Z 901.361,A -85,B 0,C 180,E1 -24865.804,E2 -24865.804} C_VEL
LIN {X 0,Y 222.357,Z 913.907,A -85,B 0,C 180,E1 -24866.302,E2 -24866.302} C_VEL
LIN {X 0,Y 219.187,Z 925.712,A -85,B 0,C 180,E1 -24866.905,E2 -24866.905} C_VEL
LIN {X 0,Y 215.945,Z 935.892,A -85,B 0,C 180,E1 -24867.522,E2 -24867.522} C_VEL
LIN {X 0,Y 211.094,Z 949.122,A -85,B 0,C 180,E1 -24868.588,E2 -24868.588} C_VEL
LIN {X 0,Y 205.585,Z 961.85,A -85,B 0,C 180,E1 -24869.838,E2 -24869.838} C_VEL
LIN {X 0,Y 200.168,Z 972.835,A -85,B 0,C 180,E1 -24871.152,E2 -24871.152} C_VEL
LIN {X 0,Y 194.278,Z 983.628,A -85,B 0,C 180,E1 -24872.749,E2 -24872.749} C_VEL
LIN {X 0,Y 187.952,Z 994.119,A -85,B 0,C 180,E1 -24874.653,E2 -24874.653} C_VEL
LIN {X 0,Y 181.753,Z 1003.379,A -85,B 0,C 180,E1 -24876.646,E2 -24876.646} C_VEL
LIN {X 0,Y 174.733,Z 1013.105,A -85,B 0,C 180,E1 -24879.264,E2 -24879.264} C_VEL
LIN {X 0,Y 168.276,Z 1021.489,A -85,B 0,C 180,E1 -24882.062,E2 -24882.062} C_VEL
LIN {X 0,Y 161.012,Z 1030.223,A -85,B 0,C 180,E1 -24885.704,E2 -24885.704} C_VEL
LIN {X 0,Y 155.438,Z 1036.654,A -85,B 0,C 180,E1 -24889.036,E2 -24889.036} C_VEL
LIN {X 0,Y 148.876,Z 1043.919,A -85,B 0,C 180,E1 -24893.838,E2 -24893.838} C_VEL
LIN {X 0,Y 144.667,Z 1048.575,A -85,B 0,C 180,E1 -24897.699,E2 -24897.699} C_VEL
LIN {X 0,Y 140.08,Z 1053.685,A -85,B 0,C 180,E1 -24903.158,E2 -24903.158} C_VEL
LIN {X 0,Y 136.707,Z 1057.699,A -85,B 0,C 180,E1 -24908.909,E2 -24908.909} C_VEL
LIN {X 0,Y 135.468,Z 1059.383,A -85,B 0,C 180,E1 -24911.864,E2 -24911.864} C_VEL
LIN {X 0,Y 133.848,Z 1061.871,A -85,B 0,C 180,E1 -24917.876,E2 -24917.876} C_VEL
LIN {X 0,Y 133.324,Z 1063.363,A -85,B 0,C 180,E1 -24923.948,E2 -24923.948} C_VEL
LIN {X 0,Y 133.533,Z 1063.869,A -85,B 0,C 180,E1 -24930,E2 -24930} C_VEL
LIN {X 0,Y 133.324,Z 1063.363,A -85,B 0,C 180,E1 -24936.052,E2 -24936.052} C_VEL
LIN {X 0,Y 134.03,Z 1061.439,A -85,B 0,C 180,E1 -24943.218,E2 -24943.218} C_VEL
LIN {X 0,Y 135.468,Z 1059.383,A -85,B 0,C 180,E1 -24948.136,E2 -24948.136} C_VEL
LIN {X 0,Y 138.253,Z 1055.868,A -85,B 0,C 180,E1 -24953.995,E2 -24953.995} C_VEL
LIN {X 0,Y 139.231,Z 1054.655,A -85,B 0,C 180,E1 -24955.586,E2 -24955.586} C_VEL
LIN {X 0,Y 140.142,Z 1052.982,A -85,B 0,C 180,E1 -24957.872,E2 -24957.872} C_VEL
LIN {X 0,Y 140.316,Z 1049.833,A -85,B 0,C 180,E1 -24961.729,E2 -24961.729} C_VEL
LIN {X 0,Y 141.045,Z 1046.487,A -85,B 0,C 180,E1 -24965.514,E2 -24965.514} C_VEL
LIN {X 0,Y 142.768,Z 1044.058,A -85,B 0,C 180,E1 -24967.592,E2 -24967.592} C_VEL
LIN {X 0,Y 148.232,Z 1038.357,A -85,B 0,C 180,E1 -24971.587,E2 -24971.587} C_VEL
LIN {X 0,Y 153.93,Z 1032.237,A -85,B 0,C 180,E1 -24975.045,E2 -24975.045} C_VEL
LIN {X 0,Y 160.162,Z 1025.256,A -85,B 0,C 180,E1 -24978.241,E2 -24978.241} C_VEL
LIN {X 0,Y 166.811,Z 1017.291,A -85,B 0,C 180,E1 -24981.207,E2 -24981.207} C_VEL
LIN {X 0,Y 173.872,Z 1008.183,A -85,B 0,C 180,E1 -24983.939,E2 -24983.939} C_VEL
LIN {X 0,Y 180.064,Z 999.622,A -85,B 0,C 180,E1 -24986.035,E2 -24986.035} C_VEL
LIN {X 0,Y 187.386,Z 988.514,A -85,B 0,C 180,E1 -24988.212,E2 -24988.212} C_VEL
LIN {X 0,Y 193.859,Z 977.612,A -85,B 0,C 180,E1 -24989.942,E2 -24989.942} C_VEL
LIN {X 0,Y 200.024,Z 965.953,A -85,B 0,C 180,E1 -24991.446,E2 -24991.446} C_VEL
LIN {X 0,Y 205.659,Z 953.939,A -85,B 0,C 180,E1 -24992.682,E2 -24992.682} C_VEL
LIN {X 0,Y 210.59,Z 941.626,A -85,B 0,C 180,E1 -24993.75,E2 -24993.75} C_VEL
LIN {X 0,Y 214.946,Z 929.092,A -85,B 0,C 180,E1 -24994.585,E2 -24994.585} C_VEL
LIN {X 0,Y 218.813,Z 915.623,A -85,B 0,C 180,E1 -24995.285,E2 -24995.285} C_VEL
LIN {X 0,Y 221.77,Z 902.866,A -85,B 0,C 180,E1 -24995.778,E2 -24995.778} C_VEL
LIN {X 0,Y 224.07,Z 888.921,A -85,B 0,C 180,E1 -24996.23,E2 -24996.23} C_VEL
LIN {X 0,Y 227.085,Z 859.511,A -85,B 0,C 180,E1 -24996.95,E2 -24996.95} C_VEL
LIN {X 0,Y 230.802,Z 819.863,A -85,B 0,C 180,E1 -24997.881,E2 -24997.881} C_VEL
LIN {X 0,Y 228.2,Z 812.346,A -85,B 0,C 180,E1 -25000.197,E2 -25000.197} C_VEL
LIN {X 0,Y 224.82,Z 805.59,A -85,B 0,C 180,E1 -25003.434,E2 -25003.434} C_VEL
LIN {X 0,Y 221.758,Z 799.929,A -85,B 0,C 180,E1 -25007.066,E2 -25007.066} C_VEL
LIN {X 0,Y 220.068,Z 796.732,A -85,B 0,C 180,E1 -25009.651,E2 -25009.651} C_VEL
LIN {X 0,Y 218.276,Z 793.061,A -85,B 0,C 180,E1 -25013.529,E2 -25013.529} C_VEL
LIN {X 0,Y 217.083,Z 790.746,A -85,B 0,C 180,E1 -25020,E2 -25020} C_VEL
LIN {X 0,Y 218.424,Z 793.353,A -85,B 0,C 180,E1 -25027.278,E2 -25027.278} C_VEL
LIN {X 0,Y 220.242,Z 796.974,A -85,B 0,C 180,E1 -25031.038,E2 -25031.038} C_VEL
LIN {X 0,Y 222.84,Z 801.862,A -85,B 0,C 180,E1 -25034.73,E2 -25034.73} C_VEL
LIN {X 0,Y 225.518,Z 806.894,A -85,B 0,C 180,E1 -25037.688,E2 -25037.688} C_VEL
LIN {X 0,Y 229.838,Z 815.681,A -85,B 0,C 180,E1 -25041.585,E2 -25041.585} C_VEL
LIN {X 0,Y 239.386,Z 834.315,A -85,B 0,C 180,E1 -25048.016,E2 -25048.016} C_VEL
LIN {X 0,Y 246.752,Z 844.5,A -85,B 0,C 180,E1 -25051.663,E2 -25051.663} C_VEL
LIN {X 0,Y 254.141,Z 852.876,A -85,B 0,C 180,E1 -25054.7,E2 -25054.7} C_VEL
LIN {X 0,Y 270.14,Z 867.468,A -85,B 0,C 180,E1 -25059.965,E2 -25059.965} C_VEL
LIN {X 0,Y 282.427,Z 876.9,A -85,B 0,C 180,E1 -25063.303,E2 -25063.303} C_VEL
LIN {X 0,Y 290.26,Z 883.015,A -85,B 0,C 180,E1 -25065.572,E2 -25065.572} C_VEL
LIN {X 0,Y 297.099,Z 888.369,A -85,B 0,C 180,E1 -25067.749,E2 -25067.749} C_VEL
LIN {X 0,Y 304.289,Z 893.806,A -85,B 0,C 180,E1 -25070.207,E2 -25070.207} C_VEL
LIN {X 0,Y 311.372,Z 899.494,A -85,B 0,C 180,E1 -25072.824,E2 -25072.824} C_VEL
LIN {X 0,Y 316.907,Z 903.88,A -85,B 0,C 180,E1 -25074.983,E2 -25074.983} C_VEL
LIN {X 0,Y 323.351,Z 908.858,A -85,B 0,C 180,E1 -25077.641,E2 -25077.641} C_VEL
LIN {X 0,Y 327.199,Z 911.741,A -85,B 0,C 180,E1 -25079.315,E2 -25079.315} C_VEL
LIN {X 0,Y 332.47,Z 915.815,A -85,B 0,C 180,E1 -25081.715,E2 -25081.715} C_VEL
LIN {X 0,Y 337.979,Z 919.597,A -85,B 0,C 180,E1 -25084.446,E2 -25084.446} C_VEL
LIN {X 0,Y 342.103,Z 922.913,A -85,B 0,C 180,E1 -25086.697,E2 -25086.697} C_VEL
LIN {X 0,Y 346.531,Z 925.941,A -85,B 0,C 180,E1 -25089.27,E2 -25089.27} C_VEL
LIN {X 0,Y 350.023,Z 928.094,A -85,B 0,C 180,E1 -25091.526,E2 -25091.526} C_VEL
LIN {X 0,Y 353.564,Z 931.148,A -85,B 0,C 180,E1 -25094.234,E2 -25094.234} C_VEL
LIN {X 0,Y 356.648,Z 933.297,A -85,B 0,C 180,E1 -25096.941,E2 -25096.941} C_VEL
LIN {X 0,Y 358.958,Z 934.632,A -85,B 0,C 180,E1 -25099.323,E2 -25099.323} C_VEL
LIN {X 0,Y 360.898,Z 935.437,A -85,B 0,C 180,E1 -25101.726,E2 -25101.726} C_VEL
LIN {X 0,Y 362.166,Z 936.025,A -85,B 0,C 180,E1 -25103.795,E2 -25103.795} C_VEL
LIN {X 0,Y 362.966,Z 936.442,A -85,B 0,C 180,E1 -25105.558,E2 -25105.558} C_VEL
LIN {X 0,Y 363.605,Z 936.642,A -85,B 0,C 180,E1 -25107.785,E2 -25107.785} C_VEL
LIN {X 0,Y 363.784,Z 936.835,A -85,B 0,C 180,E1 -25110,E2 -25110} C_VEL
LIN {X 0,Y 363.603,Z 936.641,A -85,B 0,C 180,E1 -25112.215,E2 -25112.215} C_VEL
LIN {X 0,Y 362.725,Z 936.353,A -85,B 0,C 180,E1 -25115.002,E2 -25115.002} C_VEL
LIN {X 0,Y 361.459,Z 935.698,A -85,B 0,C 180,E1 -25117.431,E2 -25117.431} C_VEL
LIN {X 0,Y 359.864,Z 935.023,A -85,B 0,C 180,E1 -25119.615,E2 -25119.615} C_VEL
LIN {X 0,Y 357.501,Z 933.817,A -85,B 0,C 180,E1 -25122.223,E2 -25122.223} C_VEL
LIN {X 0,Y 354.716,Z 932.019,A -85,B 0,C 180,E1 -25124.805,E2 -25124.805} C_VEL
LIN {X 0,Y 351.381,Z 929.283,A -85,B 0,C 180,E1 -25127.458,E2 -25127.458} C_VEL
LIN {X 0,Y 348.877,Z 927.226,A -85,B 0,C 180,E1 -25129.257,E2 -25129.257} C_VEL
LIN {X 0,Y 344.843,Z 924.863,A -85,B 0,C 180,E1 -25131.722,E2 -25131.722} C_VEL
LIN {X 0,Y 340.839,Z 921.929,A -85,B 0,C 180,E1 -25133.989,E2 -25133.989} C_VEL
LIN {X 0,Y 336.743,Z 918.601,A -85,B 0,C 180,E1 -25136.179,E2 -25136.179} C_VEL
LIN {X 0,Y 332.277,Z 915.689,A -85,B 0,C 180,E1 -25138.35,E2 -25138.35} C_VEL
LIN {X 0,Y 327.608,Z 912.053,A -85,B 0,C 180,E1 -25140.512,E2 -25140.512} C_VEL
LIN {X 0,Y 322.603,Z 908.236,A -85,B 0,C 180,E1 -25142.686,E2 -25142.686} C_VEL
LIN {X 0,Y 316.176,Z 903.257,A -85,B 0,C 180,E1 -25145.304,E2 -25145.304} C_VEL
LIN {X 0,Y 310.195,Z 898.605,A -85,B 0,C 180,E1 -25147.623,E2 -25147.623} C_VEL
LIN {X 0,Y 302.848,Z 892.761,A -85,B 0,C 180,E1 -25150.297,E2 -25150.297} C_VEL
LIN {X 0,Y 295.786,Z 887.278,A -85,B 0,C 180,E1 -25152.686,E2 -25152.686} C_VEL
LIN {X 0,Y 287.806,Z 881.134,A -85,B 0,C 180,E1 -25155.163,E2 -25155.163} C_VEL
LIN {X 0,Y 280.837,Z 875.757,A -85,B 0,C 180,E1 -25157.128,E2 -25157.128} C_VEL
LIN {X 0,Y 264.025,Z 862.163,A -85,B 0,C 180,E1 -25161.887,E2 -25161.887} C_VEL
LIN {X 0,Y 251.171,Z 849.82,A -85,B 0,C 180,E1 -25166.454,E2 -25166.454} C_VEL
LIN {X 0,Y 241.013,Z 836.783,A -85,B 0,C 180,E1 -25171.109,E2 -25171.109} C_VEL
LIN {X 0,Y 233.806,Z 824.367,A -85,B 0,C 180,E1 -25175.414,E2 -25175.414} C_VEL
LIN {X 0,Y 229.318,Z 814.683,A -85,B 0,C 180,E1 -25178.835,E2 -25178.835} C_VEL
LIN {X 0,Y 225.837,Z 807.584,A -85,B 0,C 180,E1 -25181.986,E2 -25181.986} C_VEL
LIN {X 0,Y 223.387,Z 802.948,A -85,B 0,C 180,E1 -25184.607,E2 -25184.607} C_VEL
LIN {X 0,Y 221.554,Z 799.565,A -85,B 0,C 180,E1 -25186.938,E2 -25186.938} C_VEL
LIN {X 0,Y 220.099,Z 796.763,A -85,B 0,C 180,E1 -25189.196,E2 -25189.196} C_VEL
LIN {X 0,Y 218.211,Z 792.974,A -85,B 0,C 180,E1 -25193.296,E2 -25193.296} C_VEL
LIN {X 0,Y 217.085,Z 790.729,A -85,B 0,C 180,E1 -25200,E2 -25200} C_VEL
LIN {X 0,Y 218.444,Z 793.422,A -85,B 0,C 180,E1 -25206.93,E2 -25206.93} C_VEL
LIN {X 0,Y 220.612,Z 797.742,A -85,B 0,C 180,E1 -25211.245,E2 -25211.245} C_VEL
LIN {X 0,Y 222.971,Z 802.156,A -85,B 0,C 180,E1 -25214.489,E2 -25214.489} C_VEL
LIN {X 0,Y 225.676,Z 807.227,A -85,B 0,C 180,E1 -25217.442,E2 -25217.442} C_VEL
LIN {X 0,Y 228.544,Z 813.293,A -85,B 0,C 180,E1 -25220.123,E2 -25220.123} C_VEL
LIN {X 0,Y 230.848,Z 820.03,A -85,B 0,C 180,E1 -25222.16,E2 -25222.16} C_VEL
LIN {X 0,Y 224.281,Z 887.345,A -85,B 0,C 180,E1 -25223.716,E2 -25223.716} C_VEL
LIN {X 0,Y 222.093,Z 900.995,A -85,B 0,C 180,E1 -25224.144,E2 -25224.144} C_VEL
LIN {X 0,Y 219.36,Z 913.425,A -85,B 0,C 180,E1 -25224.621,E2 -25224.621} C_VEL
LIN {X 0,Y 216.065,Z 925.506,A -85,B 0,C 180,E1 -25225.225,E2 -25225.225} C_VEL
LIN {X 0,Y 212.028,Z 937.666,A -85,B 0,C 180,E1 -25225.963,E2 -25225.963} C_VEL
LIN {X 0,Y 207.781,Z 948.916,A -85,B 0,C 180,E1 -25226.864,E2 -25226.864} C_VEL
LIN {X 0,Y 202.83,Z 960.206,A -85,B 0,C 180,E1 -25227.927,E2 -25227.927} C_VEL
LIN {X 0,Y 196.559,Z 972.628,A -85,B 0,C 180,E1 -25229.365,E2 -25229.365} C_VEL
LIN {X 0,Y 190.513,Z 983.421,A -85,B 0,C 180,E1 -25230.944,E2 -25230.944} C_VEL
LIN {X 0,Y 183.976,Z 993.912,A -85,B 0,C 180,E1 -25232.819,E2 -25232.819} C_VEL
LIN {X 0,Y 177.567,Z 1003.171,A -85,B 0,C 180,E1 -25234.79,E2 -25234.79} C_VEL
LIN {X 0,Y 170.286,Z 1012.897,A -85,B 0,C 180,E1 -25237.396,E2 -25237.396} C_VEL
LIN {X 0,Y 163.033,Z 1021.871,A -85,B 0,C 180,E1 -25240.419,E2 -25240.419} C_VEL
LIN {X 0,Y 155.958,Z 1030.016,A -85,B 0,C 180,E1 -25243.863,E2 -25243.863} C_VEL
LIN {X 0,Y 150.068,Z 1036.445,A -85,B 0,C 180,E1 -25247.231,E2 -25247.231} C_VEL
LIN {X 0,Y 142.896,Z 1043.941,A -85,B 0,C 180,E1 -25252.318,E2 -25252.318} C_VEL
LIN {X 0,Y 138.633,Z 1048.367,A -85,B 0,C 180,E1 -25256.108,E2 -25256.108} C_VEL
LIN {X 0,Y 133.686,Z 1053.476,A -85,B 0,C 180,E1 -25261.763,E2 -25261.763} C_VEL
LIN {X 0,Y 131.135,Z 1056.316,A -85,B 0,C 180,E1 -25265.658,E2 -25265.658} C_VEL
LIN {X 0,Y 128.656,Z 1059.175,A -85,B 0,C 180,E1 -25270.868,E2 -25270.868} C_VEL
LIN {X 0,Y 126.856,Z 1061.664,A -85,B 0,C 180,E1 -25277.197,E2 -25277.197} C_VEL
LIN {X 0,Y 126.231,Z 1063.157,A -85,B 0,C 180,E1 -25283.607,E2 -25283.607} C_VEL
LIN {X 0,Y 126.429,Z 1063.663,A -85,B 0,C 180,E1 -25290,E2 -25290} C_VEL
LIN {X 0,Y 126.23,Z 1063.157,A -85,B 0,C 180,E1 -25296.393,E2 -25296.393} C_VEL
LIN {X 0,Y 126.856,Z 1061.664,A -85,B 0,C 180,E1 -25302.803,E2 -25302.803} C_VEL
LIN {X 0,Y 128.656,Z 1059.175,A -85,B 0,C 180,E1 -25309.132,E2 -25309.132} C_VEL
LIN {X 0,Y 131.692,Z 1055.66,A -85,B 0,C 180,E1 -25315.273,E2 -25315.273} C_VEL
LIN {X 0,Y 135.999,Z 1051.069,A -85,B 0,C 180,E1 -25321.115,E2 -25321.115} C_VEL
LIN {X 0,Y 141.529,Z 1045.333,A -85,B 0,C 180,E1 -25326.575,E2 -25326.575} C_VEL
LIN {X 0,Y 142.768,Z 1044.058,A -85,B 0,C 180,E1 -25327.592,E2 -25327.592} C_VEL
LIN {X 0,Y 144.63,Z 1041.677,A -85,B 0,C 180,E1 -25329.602,E2 -25329.602} C_VEL
LIN {X 0,Y 148.571,Z 1032.929,A -85,B 0,C 180,E1 -25336.393,E2 -25336.393} C_VEL
LIN {X 0,Y 151.068,Z 1029.838,A -85,B 0,C 180,E1 -25338.076,E2 -25338.076} C_VEL
LIN {X 0,Y 160.035,Z 1019.93,A -85,B 0,C 180,E1 -25342.228,E2 -25342.228} C_VEL
LIN {X 0,Y 168.491,Z 1009.646,A -85,B 0,C 180,E1 -25345.465,E2 -25345.465} C_VEL
LIN {X 0,Y 176.173,Z 999.415,A -85,B 0,C 180,E1 -25347.962,E2 -25347.962} C_VEL
LIN {X 0,Y 183.217,Z 989.114,A -85,B 0,C 180,E1 -25349.973,E2 -25349.973} C_VEL
LIN {X 0,Y 190.383,Z 977.406,A -85,B 0,C 180,E1 -25351.802,E2 -25351.802} C_VEL
LIN {X 0,Y 196.71,Z 965.746,A -85,B 0,C 180,E1 -25353.274,E2 -25353.274} C_VEL
LIN {X 0,Y 202.481,Z 953.733,A -85,B 0,C 180,E1 -25354.478,E2 -25354.478} C_VEL
LIN {X 0,Y 207.539,Z 941.42,A -85,B 0,C 180,E1 -25355.513,E2 -25355.513} C_VEL
LIN {X 0,Y 211.992,Z 928.886,A -85,B 0,C 180,E1 -25356.32,E2 -25356.32} C_VEL
LIN {X 0,Y 215.97,Z 915.306,A -85,B 0,C 180,E1 -25357.001,E2 -25357.001} C_VEL
LIN {X 0,Y 218.861,Z 903.148,A -85,B 0,C 180,E1 -25357.456,E2 -25357.456} C_VEL
LIN {X 0,Y 221.303,Z 888.713,A -85,B 0,C 180,E1 -25357.913,E2 -25357.913} C_VEL
LIN {X 0,Y 224.323,Z 860.092,A -85,B 0,C 180,E1 -25358.601,E2 -25358.601} C_VEL
LIN {X 0,Y 227.888,Z 823.375,A -85,B 0,C 180,E1 -25359.432,E2 -25359.432} C_VEL
LIN {X 0,Y 226.087,Z 818.017,A -85,B 0,C 180,E1 -25361.175,E2 -25361.175} C_VEL
LIN {X 0,Y 223.211,Z 811.936,A -85,B 0,C 180,E1 -25364.125,E2 -25364.125} C_VEL
LIN {X 0,Y 220.405,Z 806.517,A -85,B 0,C 180,E1 -25367.66,E2 -25367.66} C_VEL
LIN {X 0,Y 218.93,Z 803.54,A -85,B 0,C 180,E1 -25370.064,E2 -25370.064} C_VEL
LIN {X 0,Y 217.237,Z 799.956,A -85,B 0,C 180,E1 -25373.964,E2 -25373.964} C_VEL
LIN {X 0,Y 216.212,Z 797.84,A -85,B 0,C 180,E1 -25380,E2 -25380} C_VEL
LIN {X 0,Y 217.382,Z 800.185,A -85,B 0,C 180,E1 -25386.846,E2 -25386.846} C_VEL
LIN {X 0,Y 219.487,Z 804.632,A -85,B 0,C 180,E1 -25391.31,E2 -25391.31} C_VEL
LIN {X 0,Y 221.629,Z 808.849,A -85,B 0,C 180,E1 -25394.402,E2 -25394.402} C_VEL
LIN {X 0,Y 223.865,Z 813.263,A -85,B 0,C 180,E1 -25396.998,E2 -25396.998} C_VEL
LIN {X 0,Y 227.687,Z 821.45,A -85,B 0,C 180,E1 -25400.673,E2 -25400.673} C_VEL
LIN {X 0,Y 237.174,Z 840.564,A -85,B 0,C 180,E1 -25407.394,E2 -25407.394} C_VEL
LIN {X 0,Y 244.513,Z 850.902,A -85,B 0,C 180,E1 -25411.155,E2 -25411.155} C_VEL
LIN {X 0,Y 251.689,Z 859.134,A -85,B 0,C 180,E1 -25414.193,E2 -25414.193} C_VEL
LIN {X 0,Y 261.478,Z 868.454,A -85,B 0,C 180,E1 -25417.669,E2 -25417.669} C_VEL
LIN {X 0,Y 276.874,Z 881.191,A -85,B 0,C 180,E1 -25422.205,E2 -25422.205} C_VEL
LIN {X 0,Y 284.299,Z 886.891,A -85,B 0,C 180,E1 -25424.294,E2 -25424.294} C_VEL
LIN {X 0,Y 292.396,Z 893.054,A -85,B 0,C 180,E1 -25426.772,E2 -25426.772} C_VEL
LIN {X 0,Y 299.871,Z 898.959,A -85,B 0,C 180,E1 -25429.273,E2 -25429.273} C_VEL
LIN {X 0,Y 306.462,Z 904.082,A -85,B 0,C 180,E1 -25431.625,E2 -25431.625} C_VEL
LIN {X 0,Y 313.98,Z 909.888,A -85,B 0,C 180,E1 -25434.483,E2 -25434.483} C_VEL
LIN {X 0,Y 320.12,Z 914.733,A -85,B 0,C 180,E1 -25436.987,E2 -25436.987} C_VEL
LIN {X 0,Y 324.587,Z 918.017,A -85,B 0,C 180,E1 -25438.896,E2 -25438.896} C_VEL
LIN {X 0,Y 330.33,Z 922.479,A -85,B 0,C 180,E1 -25441.509,E2 -25441.509} C_VEL
LIN {X 0,Y 335.681,Z 926.038,A -85,B 0,C 180,E1 -25444.11,E2 -25444.11} C_VEL
LIN {X 0,Y 339.728,Z 929.369,A -85,B 0,C 180,E1 -25446.306,E2 -25446.306} C_VEL
LIN {X 0,Y 344.14,Z 932.424,A -85,B 0,C 180,E1 -25448.83,E2 -25448.83} C_VEL
LIN {X 0,Y 348.266,Z 934.952,A -85,B 0,C 180,E1 -25451.421,E2 -25451.421} C_VEL
LIN {X 0,Y 351.838,Z 937.993,A -85,B 0,C 180,E1 -25454.154,E2 -25454.154} C_VEL
LIN {X 0,Y 354.768,Z 940.037,A -85,B 0,C 180,E1 -25456.687,E2 -25456.687} C_VEL
LIN {X 0,Y 357.452,Z 941.59,A -85,B 0,C 180,E1 -25459.438,E2 -25459.438} C_VEL
LIN {X 0,Y 359.526,Z 942.492,A -85,B 0,C 180,E1 -25462.135,E2 -25462.135} C_VEL
LIN {X 0,Y 360.935,Z 943.135,A -85,B 0,C 180,E1 -25464.693,E2 -25464.693} C_VEL
LIN {X 0,Y 361.655,Z 943.485,A -85,B 0,C 180,E1 -25466.658,E2 -25466.658} C_VEL
LIN {X 0,Y 362.056,Z 943.68,A -85,B 0,C 180,E1 -25468.888,E2 -25468.888} C_VEL
LIN {X 0,Y 362.053,Z 943.675,A -85,B 0,C 180,E1 -25471.112,E2 -25471.112} C_VEL
LIN {X 0,Y 361.647,Z 943.495,A -85,B 0,C 180,E1 -25473.342,E2 -25473.342} C_VEL
LIN {X 0,Y 360.826,Z 943.084,A -85,B 0,C 180,E1 -25475.589,E2 -25475.589} C_VEL
LIN {X 0,Y 359.517,Z 942.511,A -85,B 0,C 180,E1 -25477.865,E2 -25477.865} C_VEL
LIN {X 0,Y 357.762,Z 941.703,A -85,B 0,C 180,E1 -25480.183,E2 -25480.183} C_VEL
LIN {X 0,Y 355.372,Z 940.444,A -85,B 0,C 180,E1 -25482.744,E2 -25482.744} C_VEL
LIN {X 0,Y 352.452,Z 938.451,A -85,B 0,C 180,E1 -25485.354,E2 -25485.354} C_VEL
LIN {X 0,Y 348.956,Z 935.556,A -85,B 0,C 180,E1 -25488.068,E2 -25488.068} C_VEL
LIN {X 0,Y 346.86,Z 933.955,A -85,B 0,C 180,E1 -25489.519,E2 -25489.519} C_VEL
LIN {X 0,Y 342.476,Z 931.313,A -85,B 0,C 180,E1 -25492.141,E2 -25492.141} C_VEL
LIN {X 0,Y 338.108,Z 928.104,A -85,B 0,C 180,E1 -25494.564,E2 -25494.564} C_VEL
LIN {X 0,Y 334.378,Z 925.133,A -85,B 0,C 180,E1 -25496.534,E2 -25496.534} C_VEL
LIN {X 0,Y 329.569,Z 921.964,A -85,B 0,C 180,E1 -25498.83,E2 -25498.83} C_VEL
LIN {X 0,Y 324.366,Z 917.774,A -85,B 0,C 180,E1 -25501.202,E2 -25501.202} C_VEL
LIN {X 0,Y 317.316,Z 912.658,A -85,B 0,C 180,E1 -25504.154,E2 -25504.154} C_VEL
LIN {X 0,Y 310.144,Z 906.902,A -85,B 0,C 180,E1 -25507.002,E2 -25507.002} C_VEL
LIN {X 0,Y 303.212,Z 901.434,A -85,B 0,C 180,E1 -25509.551,E2 -25509.551} C_VEL
LIN {X 0,Y 295.608,Z 895.679,A -85,B 0,C 180,E1 -25512.17,E2 -25512.17} C_VEL
LIN {X 0,Y 288.125,Z 889.768,A -85,B 0,C 180,E1 -25514.568,E2 -25514.568} C_VEL
LIN {X 0,Y 280.737,Z 883.984,A -85,B 0,C 180,E1 -25516.741,E2 -25516.741} C_VEL
LIN {X 0,Y 270.784,Z 876.313,A -85,B 0,C 180,E1 -25519.484,E2 -25519.484} C_VEL
LIN {X 0,Y 255.073,Z 862.649,A -85,B 0,C 180,E1 -25524.527,E2 -25524.527} C_VEL
LIN {X 0,Y 245.04,Z 851.581,A -85,B 0,C 180,E1 -25528.602,E2 -25528.602} C_VEL
LIN {X 0,Y 238.077,Z 841.929,A -85,B 0,C 180,E1 -25532.099,E2 -25532.099} C_VEL
LIN {X 0,Y 231.407,Z 829.941,A -85,B 0,C 180,E1 -25536.331,E2 -25536.331} C_VEL
LIN {X 0,Y 227.249,Z 820.5,A -85,B 0,C 180,E1 -25539.711,E2 -25539.711} C_VEL
LIN {X 0,Y 223.764,Z 813.045,A -85,B 0,C 180,E1 -25543.111,E2 -25543.111} C_VEL
LIN {X 0,Y 220.92,Z 807.363,A -85,B 0,C 180,E1 -25546.549,E2 -25546.549} C_VEL
LIN {X 0,Y 218.895,Z 803.532,A -85,B 0,C 180,E1 -25549.709,E2 -25549.709} C_VEL
LIN {X 0,Y 217.26,Z 799.963,A -85,B 0,C 180,E1 -25553.5,E2 -25553.5} C_VEL
LIN {X 0,Y 216.215,Z 797.815,A -85,B 0,C 180,E1 -25560,E2 -25560} C_VEL
LIN {X 0,Y 217.399,Z 800.251,A -85,B 0,C 180,E1 -25566.497,E2 -25566.497} C_VEL
LIN {X 0,Y 219.382,Z 804.451,A -85,B 0,C 180,E1 -25570.732,E2 -25570.732} C_VEL
LIN {X 0,Y 221.623,Z 808.878,A -85,B 0,C 180,E1 -25573.993,E2 -25573.993} C_VEL
LIN {X 0,Y 224.05,Z 813.66,A -85,B 0,C 180,E1 -25576.79,E2 -25576.79} C_VEL
LIN {X 0,Y 226.523,Z 819.145,A -85,B 0,C 180,E1 -25579.248,E2 -25579.248} C_VEL
LIN {X 0,Y 227.894,Z 823.387,A -85,B 0,C 180,E1 -25580.574,E2 -25580.574} C_VEL
LIN {X 0,Y 221.491,Z 887.316,A -85,B 0,C 180,E1 -25582.034,E2 -25582.034} C_VEL
LIN {X 0,Y 219.297,Z 900.728,A -85,B 0,C 180,E1 -25582.448,E2 -25582.448} C_VEL
LIN {X 0,Y 216.607,Z 912.82,A -85,B 0,C 180,E1 -25582.9,E2 -25582.9} C_VEL
LIN {X 0,Y 213.134,Z 925.301,A -85,B 0,C 180,E1 -25583.497,E2 -25583.497} C_VEL
LIN {X 0,Y 209.017,Z 937.461,A -85,B 0,C 180,E1 -25584.213,E2 -25584.213} C_VEL
LIN {X 0,Y 204.662,Z 948.71,A -85,B 0,C 180,E1 -25585.085,E2 -25585.085} C_VEL
LIN {X 0,Y 199.587,Z 960,A -85,B 0,C 180,E1 -25586.117,E2 -25586.117} C_VEL
LIN {X 0,Y 193.169,Z 972.422,A -85,B 0,C 180,E1 -25587.526,E2 -25587.526} C_VEL
LIN {X 0,Y 186.935,Z 983.214,A -85,B 0,C 180,E1 -25589.063,E2 -25589.063} C_VEL
LIN {X 0,Y 180.2,Z 993.705,A -85,B 0,C 180,E1 -25590.907,E2 -25590.907} C_VEL
LIN {X 0,Y 173.563,Z 1002.963,A -85,B 0,C 180,E1 -25592.839,E2 -25592.839} C_VEL
LIN {X 0,Y 166.021,Z 1012.689,A -85,B 0,C 180,E1 -25595.426,E2 -25595.426} C_VEL
LIN {X 0,Y 158.707,Z 1021.367,A -85,B 0,C 180,E1 -25598.314,E2 -25598.314} C_VEL
LIN {X 0,Y 151.079,Z 1029.808,A -85,B 0,C 180,E1 -25601.903,E2 -25601.903} C_VEL
LIN {X 0,Y 144.843,Z 1036.236,A -85,B 0,C 180,E1 -25605.288,E2 -25605.288} C_VEL
LIN {X 0,Y 138.263,Z 1042.755,A -85,B 0,C 180,E1 -25609.682,E2 -25609.682} C_VEL
LIN {X 0,Y 132.694,Z 1048.158,A -85,B 0,C 180,E1 -25614.367,E2 -25614.367} C_VEL
LIN {X 0,Y 127.366,Z 1053.267,A -85,B 0,C 180,E1 -25620.225,E2 -25620.225} C_VEL
LIN {X 0,Y 123.379,Z 1057.283,A -85,B 0,C 180,E1 -25626.501,E2 -25626.501} C_VEL
LIN {X 0,Y 120.682,Z 1060.258,A -85,B 0,C 180,E1 -25633.072,E2 -25633.072} C_VEL
LIN {X 0,Y 119.872,Z 1061.457,A -85,B 0,C 180,E1 -25636.437,E2 -25636.437} C_VEL
LIN {X 0,Y 119.159,Z 1062.951,A -85,B 0,C 180,E1 -25643.226,E2 -25643.226} C_VEL
LIN {X 0,Y 119.334,Z 1063.458,A -85,B 0,C 180,E1 -25650,E2 -25650} C_VEL
LIN {X 0,Y 119.159,Z 1062.951,A -85,B 0,C 180,E1 -25656.774,E2 -25656.774} C_VEL
